ABB RAPID module: TCTM800_DATA.mod

MODULE TCTM800_DATA
    !***********************************************************
    ! Project: P21-100538
    ! Description:
    !   Routines/functions can be modified for the customer
    !
    ! Author: RLZ
    ! Version: 1.0
    ! Date: 04-2022
    !***********************************************************
    !
    !Software axis block
    !Axis 1:                       (-90,-90)
    !Axis 3:                       (-80)
    !
    CONST string sProject:="P21-100538";
    CONST string sScreenMaker:="TpsViewHMI_6700_130220.gtpu.dll";
    !
    CONST num MAX_SPEED:=1000;
    !
    CONST pos WZ_Robot_Home_Box_MIN:=[0,600,1600];
    CONST pos WZ_Robot_Home_Box_MAX:=[800,1600,3000];
    !
    CONST pos WZ_Robot_Inside_Reach_MIN:=[-5000,-5000,-5000];
    CONST pos WZ_Robot_Inside_Reach_MAX:=[15000,5000,5000];
    !
    PERS speeddata vHighSpeed:=[4000,500,150,1000];
    PERS speeddata vHomeBoxSpeed:=[400,80,150,1000];
    PERS speeddata vLowSpeed:=[1000,500,150,1000];
    PERS speeddata vSlowSpeed:=[500,50,150,1000];
    PERS speeddata vSearchSpeed:=[250,500,150,1000];
    PERS speeddata vXsSlowSpeed:=[100,500,150,1000];
    PERS speeddata vXXsSlowSpeed:=[50,500,150,1000];
    !
!    PERS robtarget TargetNew{4000};
    PERS robtarget TargetNew{4000}:=[  [[-19.8208,13.3822,35.1781],[0.985491,-0.093353,0.141246,-0.0119022],[-1,2,-1,1],[6236.68,9E+09,9E+09,9E+09,9E+09,9E+09]],
                                        [[-19.8238,14.3776,34.9882],[0.985491,-0.093353,0.141246,-0.0119022],[-1,2,-1,1],[6236.68,9E+09,9E+09,9E+09,9E+09,9E+09]],
                                        [[-19.8267,15.373,34.7984],[0.985491,-0.093353,0.141246,-0.0119022],[-1,2,-1,1],[6236.68,9E+09,9E+09,9E+09,9E+09,9E+09]],
                                        [[-19.8297,16.3684,34.6085],[0.985491,-0.093353,0.141246,-0.0119022],[-1,2,-1,1],[6236.68,9E+09,9E+09,9E+09,9E+09,9E+09]],
                                        [[-19.8326,17.3638,34.4186],[0.985491,-0.093353,0.141246,-0.0119022],[-1,2,-1,1],[6236.68,9E+09,9E+09,9E+09,9E+09,9E+09]],
                                        [[-19.8356,18.3591,34.2288],[0.985491,-0.093353,0.141246,-0.0119022],[-1,2,-1,1],[6236.68,9E+09,9E+09,9E+09,9E+09,9E+09]],
                                        [[-19.8385,19.3545,34.0389],[0.985491,-0.093353,0.141246,-0.0119022],[-1,2,-1,1],[6236.68,9E+09,9E+09,9E+09,9E+09,9E+09]],
                                        [[-19.8415,20.3499,33.8491],[0.985491,-0.093353,0.141246,-0.0119022],[-1,2,-1,1],[6236.68,9E+09,9E+09,9E+09,9E+09,9E+09]],
                                        [[-19.8444,21.3453,33.6592],[0.985491,-0.093353,0.141246,-0.0119022],[-1,2,-1,1],[6236.68,9E+09,9E+09,9E+09,9E+09,9E+09]],
                                        [[-19.8474,22.3407,33.4694],[0.985491,-0.093353,0.141246,-0.0119022],[-1,2,-1,1],[6236.68,9E+09,9E+09,9E+09,9E+09,9E+09]],
                                        [[-19.8503,23.3361,33.2795],[0.985491,-0.093353,0.141246,-0.0119022],[-1,2,-1,1],[6236.68,9E+09,9E+09,9E+09,9E+09,9E+09]],
                                        [[-19.8533,24.3315,33.0896],[0.985491,-0.093353,0.141246,-0.0119022],[-1,2,-1,1],[6236.68,9E+09,9E+09,9E+09,9E+09,9E+09]],
                                        [[-19.8562,25.3268,32.8998],[0.985491,-0.093353,0.141246,-0.0119022],[-1,2,-1,1],[6236.68,9E+09,9E+09,9E+09,9E+09,9E+09]],
                                        [[-19.8592,26.3222,32.7099],[0.985491,-0.093353,0.141246,-0.0119022],[-1,2,-1,1],[6236.68,9E+09,9E+09,9E+09,9E+09,9E+09]],
                                        [[-19.8621,27.3176,32.5201],[0.985491,-0.093353,0.141246,-0.0119022],[-1,2,-1,1],[6236.68,9E+09,9E+09,9E+09,9E+09,9E+09]],
                                        [[-19.8651,28.313,32.3302],[0.985491,-0.093353,0.141246,-0.0119022],[-1,2,-1,1],[6236.68,9E+09,9E+09,9E+09,9E+09,9E+09]],
                                        [[-19.868,29.3084,32.1403],[0.985491,-0.093353,0.141246,-0.0119022],[-1,2,-1,1],[6236.68,9E+09,9E+09,9E+09,9E+09,9E+09]],
                                        [[-19.871,30.3038,31.9505],[0.985491,-0.093353,0.141246,-0.0119022],[-1,2,-1,1],[6236.68,9E+09,9E+09,9E+09,9E+09,9E+09]],
                                        [[-19.8739,31.2992,31.7606],[0.985491,-0.093353,0.141246,-0.0119022],[-1,2,-1,1],[6236.68,9E+09,9E+09,9E+09,9E+09,9E+09]],
                                        [[-19.8769,32.2945,31.5708],[0.985491,-0.093353,0.141246,-0.0119022],[-1,2,-1,1],[6236.68,9E+09,9E+09,9E+09,9E+09,9E+09]],
                                        [[-19.8798,33.2899,31.3809],[0.985491,-0.093353,0.141246,-0.0119022],[-1,2,-1,1],[6236.68,9E+09,9E+09,9E+09,9E+09,9E+09]],
                                        [[-19.8828,34.2853,31.1911],[0.985491,-0.093353,0.141246,-0.0119022],[-1,2,-1,1],[6236.68,9E+09,9E+09,9E+09,9E+09,9E+09]],
                                        [[-19.8857,35.2807,31.0012],[0.985675,-0.0933685,0.139955,-0.01178],[-1,2,-1,1],[6234.68,9E+09,9E+09,9E+09,9E+09,9E+09]],
                                        [[-19.8887,36.2761,30.8113],[0.985675,-0.0933685,0.139955,-0.01178],[-1,2,-1,1],[6232.68,9E+09,9E+09,9E+09,9E+09,9E+09]],
                                        [[-19.8916,37.2715,30.6215],[0.985675,-0.0933685,0.139955,-0.01178],[-1,2,-1,1],[6230.68,9E+09,9E+09,9E+09,9E+09,9E+09]],
                                        [[-19.8946,38.2669,30.4316],[0.985675,-0.0933685,0.139955,-0.01178],[-1,2,-1,1],[6228.68,9E+09,9E+09,9E+09,9E+09,9E+09]],
                                        [[-19.8976,39.2622,30.2418],[0.985675,-0.0933685,0.139955,-0.01178],[-1,2,-1,1],[6226.68,9E+09,9E+09,9E+09,9E+09,9E+09]],
                                        [[-19.9005,40.2576,30.0519],[0.985675,-0.0933685,0.139955,-0.01178],[-1,2,-1,1],[6224.68,9E+09,9E+09,9E+09,9E+09,9E+09]],
                                        [[-19.9035,41.253,29.8621],[0.985675,-0.0933685,0.139955,-0.01178],[-1,2,-1,1],[6222.68,9E+09,9E+09,9E+09,9E+09,9E+09]],
                                        [[-19.9064,42.2484,29.6722],[0.985675,-0.0933685,0.139955,-0.01178],[-1,2,-1,1],[6220.68,9E+09,9E+09,9E+09,9E+09,9E+09]],
                                        [[-19.9094,43.2438,29.4823],[0.985675,-0.0933685,0.139955,-0.01178],[-1,2,-1,1],[6218.68,9E+09,9E+09,9E+09,9E+09,9E+09]],
                                        [[-19.9123,44.2392,29.2925],[0.985675,-0.0933685,0.139955,-0.01178],[-1,2,-1,1],[6216.68,9E+09,9E+09,9E+09,9E+09,9E+09]],
                                        [[-19.9153,45.2346,29.1026],[0.985675,-0.0933685,0.139955,-0.01178],[-1,2,-1,1],[6214.68,9E+09,9E+09,9E+09,9E+09,9E+09]],
                                        [[-19.9182,46.2299,28.9128],[0.985675,-0.0933685,0.139955,-0.01178],[-1,2,-1,1],[6212.68,9E+09,9E+09,9E+09,9E+09,9E+09]],
                                        [[-19.9212,47.2253,28.7229],[0.985675,-0.0933685,0.139955,-0.01178],[-1,2,-1,1],[6210.68,9E+09,9E+09,9E+09,9E+09,9E+09]],
                                        [[-19.9241,48.2207,28.533],[0.929993,-0.0883232,0.355355,-0.0321736],[-1,2,-1,1],[6212.68,9E+09,9E+09,9E+09,9E+09,9E+09]],
                                        [[-19.9271,49.2161,28.3432],[0.930471,-0.0882227,0.354142,-0.0319903],[-1,2,-1,1],[6214.68,9E+09,9E+09,9E+09,9E+09,9E+09]],
                                        [[-19.93,50.2115,28.1533],[0.930952,-0.0880818,0.352929,-0.031787],[-1,2,-1,1],[6216.68,9E+09,9E+09,9E+09,9E+09,9E+09]],
                                        [[-19.933,51.2069,27.9635],[0.931436,-0.0879018,0.351717,-0.0315633],[-1,2,-1,1],[6218.68,9E+09,9E+09,9E+09,9E+09,9E+09]],
                                        [[-19.9359,52.2022,27.7736],[0.931921,-0.0876857,0.350504,-0.0313225],[-1,2,-1,1],[6220.68,9E+09,9E+09,9E+09,9E+09,9E+09]],
                                        [[-19.9389,53.1976,27.5838],[0.932407,-0.0874409,0.349293,-0.0310697],[-1,2,-1,1],[6222.68,9E+09,9E+09,9E+09,9E+09,9E+09]],
                                        [[-19.9418,54.193,27.3939],[0.932894,-0.0871662,0.348081,-0.0308115],[-1,2,-1,1],[6224.68,9E+09,9E+09,9E+09,9E+09,9E+09]],
                                        [[-19.9448,55.1884,27.204],[0.933381,-0.0868686,0.346871,-0.0305526],[-1,2,-1,1],[6226.68,9E+09,9E+09,9E+09,9E+09,9E+09]],
                                        [[-19.9477,56.1838,27.0142],[0.933868,-0.0865579,0.34566,-0.0302899],[-1,2,-1,1],[6228.68,9E+09,9E+09,9E+09,9E+09,9E+09]],
                                        [[-19.9507,57.1792,26.8243],[0.934353,-0.0862461,0.344448,-0.0300257],[-1,2,-1,1],[6230.68,9E+09,9E+09,9E+09,9E+09,9E+09]],
                                        [[-19.9536,58.1746,26.6345],[0.934837,-0.0859295,0.343235,-0.0297506],[-1,2,-1,1],[6232.68,9E+09,9E+09,9E+09,9E+09,9E+09]],
                                        [[-19.9566,59.1699,26.4446],[0.93532,-0.0856102,0.342021,-0.0294673],[-1,2,-1,1],[6234.68,9E+09,9E+09,9E+09,9E+09,9E+09]],
                                        [[-19.9595,60.1653,26.2548],[0.935802,-0.0852947,0.340805,-0.0291789],[-1,2,-1,1],[6236.68,9E+09,9E+09,9E+09,9E+09,9E+09]],
                                        [[-19.9625,61.1607,26.0649],[0.936281,-0.0849877,0.339588,-0.0288886],[-1,2,-1,1],[6238.68,9E+09,9E+09,9E+09,9E+09,9E+09]],
                                        [[-19.9654,62.1561,25.875],[0.936758,-0.0846954,0.33837,-0.0285976],[-1,2,-1,1],[6240.68,9E+09,9E+09,9E+09,9E+09,9E+09]],
                                        [[-19.9684,63.1515,25.6852],[0.937231,-0.0844174,0.33715,-0.0283113],[-1,2,-1,1],[6242.68,9E+09,9E+09,9E+09,9E+09,9E+09]],
                                        [[-19.9713,64.1469,25.4953],[0.937701,-0.0841591,0.335928,-0.0280356],[-1,2,-1,1],[6244.68,9E+09,9E+09,9E+09,9E+09,9E+09]],
                                        [[-19.9792,65.5555,25.2738],[0.938167,-0.0839191,0.334706,-0.0277747],[-1,2,-1,1],[6246.68,9E+09,9E+09,9E+09,9E+09,9E+09]],
                                        [[-19.9846,66.7312,25.0742],[0.938629,-0.0837057,0.333483,-0.0275222],[-1,2,-1,1],[6248.68,9E+09,9E+09,9E+09,9E+09,9E+09]],
                                        [[-19.9903,67.8868,24.8779],[0.939087,-0.0835199,0.332257,-0.0272796],[-1,2,-1,1],[6250.68,9E+09,9E+09,9E+09,9E+09,9E+09]],
                                        [[-19.9968,69.025,24.6862],[0.939537,-0.0834029,0.33103,-0.0270736],[-1,2,-1,1],[6252.68,9E+09,9E+09,9E+09,9E+09,9E+09]],
                                        [[-20.0023,70.1507,24.4974],[0.939978,-0.0833611,0.3298,-0.0269014],[-1,2,-1,1],[6254.68,9E+09,9E+09,9E+09,9E+09,9E+09]],
                                        [[-20.0074,71.2662,24.3079],[0.940411,-0.0833921,0.328567,-0.026763],[-1,2,-1,1],[6256.68,9E+09,9E+09,9E+09,9E+09,9E+09]],
                                        [[-20.0097,72.3751,24.121],[0.940835,-0.0835,0.327332,-0.0266604],[-1,2,-1,1],[6258.68,9E+09,9E+09,9E+09,9E+09,9E+09]],
                                        [[-20.0112,73.4816,23.9325],[0.94125,-0.0836821,0.326095,-0.0265903],[-1,2,-1,1],[6260.68,9E+09,9E+09,9E+09,9E+09,9E+09]],
                                        [[-20.0151,74.5864,23.7424],[0.941657,-0.0839444,0.324855,-0.0265527],[-1,2,-1,1],[6262.68,9E+09,9E+09,9E+09,9E+09,9E+09]],
                                        [[-20.0203,75.6949,23.5472],[0.942055,-0.0842785,0.323612,-0.0265474],[-1,2,-1,1],[6264.68,9E+09,9E+09,9E+09,9E+09,9E+09]],
                                        [[-20.0287,76.8065,23.3556],[0.942445,-0.084682,0.322367,-0.0265724],[-1,2,-1,1],[6266.68,9E+09,9E+09,9E+09,9E+09,9E+09]],
                                        [[-20.0368,77.9219,23.1634],[0.942828,-0.0851371,0.321121,-0.0266187],[-1,2,-1,1],[6268.68,9E+09,9E+09,9E+09,9E+09,9E+09]],
                                        [[-20.0447,79.0403,22.9681],[0.943204,-0.0856504,0.319872,-0.0266856],[-1,2,-1,1],[6270.68,9E+09,9E+09,9E+09,9E+09,9E+09]],
                                        [[-20.0527,80.1618,22.7711],[0.943573,-0.0862256,0.31862,-0.0267765],[-1,2,-1,1],[6272.68,9E+09,9E+09,9E+09,9E+09,9E+09]],
                                        [[-20.0612,81.2846,22.5719],[0.943932,-0.0868722,0.317367,-0.0269036],[-1,2,-1,1],[6274.68,9E+09,9E+09,9E+09,9E+09,9E+09]],
                                        [[-20.0679,82.4167,22.3707],[0.944282,-0.0875917,0.316112,-0.0270609],[-1,2,-1,1],[6276.68,9E+09,9E+09,9E+09,9E+09,9E+09]],
                                        [[-20.0726,83.5525,22.1667],[0.944623,-0.0883798,0.314854,-0.0272472],[-1,2,-1,1],[6278.68,9E+09,9E+09,9E+09,9E+09,9E+09]],
                                        [[-20.0759,84.6909,21.9623],[0.944955,-0.0892357,0.313595,-0.027466],[-1,2,-1,1],[6280.49,9E+09,9E+09,9E+09,9E+09,9E+09]],
                                        [[-20.0829,85.8322,21.7552],[0.945292,-0.090032,0.312336,-0.0276392],[-1,2,-1,1],[6282.04,9E+09,9E+09,9E+09,9E+09,9E+09]],
                                        [[-20.0895,86.9766,21.5476],[0.94563,-0.0908122,0.311073,-0.0277661],[-1,2,-1,1],[6283.36,9E+09,9E+09,9E+09,9E+09,9E+09]],
                                        [[-20.09,87.9047,21.3558],[0.94597,-0.0915639,0.309808,-0.0278434],[-1,2,-1,1],[6284.46,9E+09,9E+09,9E+09,9E+09,9E+09]],
                                        [[-20.0924,88.8463,21.1574],[0.946315,-0.0922771,0.30854,-0.0278587],[-1,2,-1,1],[6285.55,9E+09,9E+09,9E+09,9E+09,9E+09]],
                                        [[-20.0944,89.8013,20.9561],[0.946663,-0.0929378,0.307272,-0.0278381],[-1,2,-1,1],[6286.4,9E+09,9E+09,9E+09,9E+09,9E+09]],
                                        [[-20.0959,90.781,20.7473],[0.947015,-0.0935522,0.306003,-0.0277818],[-1,2,-1,1],[6287.04,9E+09,9E+09,9E+09,9E+09,9E+09]],
                                        [[-20.0983,91.779,20.5356],[0.947371,-0.0941184,0.304734,-0.027689],[-1,2,-1,1],[6287.46,9E+09,9E+09,9E+09,9E+09,9E+09]],
                                        [[-20.1012,92.7833,20.3188],[0.947729,-0.0946464,0.303465,-0.0275732],[-1,2,-1,1],[6287.67,9E+09,9E+09,9E+09,9E+09,9E+09]],
                                        [[-20.1031,93.793,20.1035],[0.94809,-0.0951344,0.302195,-0.0274276],[-1,2,-1,1],[6287.7,9E+09,9E+09,9E+09,9E+09,9E+09]],
                                        [[-20.1053,94.8139,19.887],[0.948456,-0.0955701,0.300925,-0.0272494],[-1,2,-1,1],[6287.54,9E+09,9E+09,9E+09,9E+09,9E+09]],
                                        [[-20.1085,95.8306,19.6795],[0.948826,-0.0959528,0.299654,-0.0270214],[-1,2,-1,1],[6287.21,9E+09,9E+09,9E+09,9E+09,9E+09]],
                                        [[-20.113,96.8463,19.469],[0.949202,-0.0962697,0.298382,-0.026743],[-1,2,-1,1],[6286.72,9E+09,9E+09,9E+09,9E+09,9E+09]],
                                        [[-20.1163,97.8528,19.258],[0.949586,-0.0965149,0.297109,-0.0264101],[-1,2,-1,1],[6286.07,9E+09,9E+09,9E+09,9E+09,9E+09]],
                                        [[-20.1158,98.8519,19.0415],[0.949976,-0.0966895,0.295836,-0.0260264],[-1,2,-1,1],[6285.28,9E+09,9E+09,9E+09,9E+09,9E+09]],
                                        [[-20.118,99.846,18.8262],[0.950371,-0.0968106,0.294562,-0.0255972],[-1,2,-1,1],[6284.35,9E+09,9E+09,9E+09,9E+09,9E+09]],
                                        [[-20.1194,100.834,18.6136],[0.950772,-0.0968625,0.293289,-0.0251351],[-1,2,-1,1],[6283.29,9E+09,9E+09,9E+09,9E+09,9E+09]],
                                        [[-20.1198,101.816,18.4019],[0.95118,-0.0968264,0.292018,-0.0246466],[-1,2,-1,1],[6282.1,9E+09,9E+09,9E+09,9E+09,9E+09]],
                                        [[-20.132,102.941,18.1808],[0.951594,-0.0967003,0.290751,-0.0241347],[-1,2,-1,1],[6280.79,9E+09,9E+09,9E+09,9E+09,9E+09]],
                                        [[-20.1525,104.034,17.9652],[0.952015,-0.0964822,0.289486,-0.0236033],[-1,2,-1,1],[6279.23,9E+09,9E+09,9E+09,9E+09,9E+09]],
                                        [[-20.1727,105.104,17.7578],[0.952442,-0.096171,0.288226,-0.0230543],[-1,2,-1,1],[6277.6,9E+09,9E+09,9E+09,9E+09,9E+09]],
                                        [[-20.1965,106.149,17.558],[0.95287,-0.0958206,0.286967,-0.0225081],[-1,2,-1,1],[6275.89,9E+09,9E+09,9E+09,9E+09,9E+09]],
                                        [[-20.2098,107.165,17.3633],[0.953295,-0.0954673,0.285711,-0.0219992],[-1,2,-1,1],[6274.12,9E+09,9E+09,9E+09,9E+09,9E+09]],
                                        [[-20.2242,108.185,17.1667],[0.953715,-0.0951127,0.284459,-0.0215388],[-1,2,-1,1],[6272.29,9E+09,9E+09,9E+09,9E+09,9E+09]],
                                        [[-20.2425,109.218,16.9643],[0.954131,-0.0947572,0.28321,-0.0211306],[-1,2,-1,1],[6270.39,9E+09,9E+09,9E+09,9E+09,9E+09]],
                                        [[-20.2581,110.254,16.7562],[0.954543,-0.0944062,0.281965,-0.0207777],[-1,2,-1,1],[6268.41,9E+09,9E+09,9E+09,9E+09,9E+09]],
                                        [[-20.2753,111.299,16.547],[0.954949,-0.0940667,0.280722,-0.0204648],[-1,2,-1,1],[6266.41,9E+09,9E+09,9E+09,9E+09,9E+09]],
                                        [[-20.2912,112.342,16.3468],[0.955352,-0.09373,0.279481,-0.0201944],[-1,2,-1,1],[6264.41,9E+09,9E+09,9E+09,9E+09,9E+09]],
                                        [[-20.3116,113.385,16.1428],[0.955753,-0.0933758,0.278243,-0.0199595],[-1,2,-1,1],[6262.41,9E+09,9E+09,9E+09,9E+09,9E+09]],
                                        [[-20.3318,114.437,15.9409],[0.956155,-0.0929712,0.27701,-0.0197528],[-1,2,-1,1],[6260.41,9E+09,9E+09,9E+09,9E+09,9E+09]],
                                        [[-20.3539,115.497,15.7419],[0.956556,-0.0925336,0.275781,-0.0195746],[-1,2,-1,1],[6258.41,9E+09,9E+09,9E+09,9E+09,9E+09]],
                                        [[-20.376,116.553,15.5421],[0.956956,-0.0920778,0.274554,-0.0194295],[-1,2,-1,1],[6256.41,9E+09,9E+09,9E+09,9E+09,9E+09]],
                                        [[-20.3986,117.615,15.334],[0.957352,-0.0916118,0.273332,-0.0193503],[-1,2,-1,1],[6254.41,9E+09,9E+09,9E+09,9E+09,9E+09]],
                                        [[-20.4172,118.682,15.1287],[0.957744,-0.0911493,0.272113,-0.0193238],[-1,2,-1,1],[6252.41,9E+09,9E+09,9E+09,9E+09,9E+09]],
                                        [[-20.4343,119.758,14.9301],[0.958131,-0.0906871,0.270898,-0.0193504],[-1,2,-1,1],[6250.41,9E+09,9E+09,9E+09,9E+09,9E+09]],
                                        [[-20.4523,120.845,14.7299],[0.958515,-0.0902277,0.269686,-0.0194368],[-1,2,-1,1],[6248.41,9E+09,9E+09,9E+09,9E+09,9E+09]],
                                        [[-20.4663,121.94,14.5304],[0.958898,-0.089739,0.268477,-0.0195467],[-1,2,-1,1],[6246.41,9E+09,9E+09,9E+09,9E+09,9E+09]],
                                        [[-20.4807,123.047,14.3291],[0.959282,-0.0892157,0.267268,-0.0196568],[-1,2,-1,1],[6244.41,9E+09,9E+09,9E+09,9E+09,9E+09]],
                                        [[-20.4981,124.154,14.1317],[0.959667,-0.0886629,0.266059,-0.0197558],[-1,2,-1,1],[6242.41,9E+09,9E+09,9E+09,9E+09,9E+09]],
                                        [[-20.5026,125.121,13.9475],[0.960055,-0.0880643,0.26485,-0.0198288],[-1,2,-1,1],[6240.41,9E+09,9E+09,9E+09,9E+09,9E+09]],
                                        [[-20.5034,126.11,13.7579],[0.960445,-0.087429,0.263639,-0.0198882],[-1,2,-1,1],[6238.41,9E+09,9E+09,9E+09,9E+09,9E+09]],
                                        [[-20.5034,127.127,13.5658],[0.960836,-0.0867591,0.262429,-0.0199342],[-1,2,-1,1],[6236.41,9E+09,9E+09,9E+09,9E+09,9E+09]],
                                        [[-20.5024,128.169,13.3659],[0.961228,-0.0860689,0.261217,-0.0199642],[-1,2,-1,1],[6234.41,9E+09,9E+09,9E+09,9E+09,9E+09]],
                                        [[-20.5079,129.246,13.1642],[0.961619,-0.0853668,0.260003,-0.0199849],[-1,2,-1,1],[6232.41,9E+09,9E+09,9E+09,9E+09,9E+09]],
                                        [[-20.5129,130.318,12.9654],[0.96201,-0.0846451,0.258789,-0.0200034],[-1,2,-1,1],[6230.41,9E+09,9E+09,9E+09,9E+09,9E+09]],
                                        [[-20.5176,131.386,12.7781],[0.962402,-0.0838952,0.257574,-0.0200107],[-1,2,-1,1],[6228.41,9E+09,9E+09,9E+09,9E+09,9E+09]],
                                        [[-20.521,132.452,12.6002],[0.962793,-0.083134,0.256357,-0.0199986],[-1,2,-1,1],[6226.41,9E+09,9E+09,9E+09,9E+09,9E+09]],
                                        [[-20.5242,133.524,12.4195],[0.963184,-0.0823558,0.255137,-0.0199609],[-1,2,-1,1],[6224.41,9E+09,9E+09,9E+09,9E+09,9E+09]],
                                        [[-20.529,134.597,12.236],[0.963577,-0.0815547,0.253915,-0.0198901],[-1,2,-1,1],[6222.41,9E+09,9E+09,9E+09,9E+09,9E+09]],
                                        [[-20.5243,135.676,12.0539],[0.963969,-0.0807422,0.25269,-0.019793],[-1,2,-1,1],[6220.41,9E+09,9E+09,9E+09,9E+09,9E+09]],
                                        [[-20.5241,136.752,11.8701],[0.964361,-0.0799295,0.251461,-0.0196632],[-1,2,-1,1],[6218.41,9E+09,9E+09,9E+09,9E+09,9E+09]],
                                        [[-20.5233,137.834,11.6876],[0.964753,-0.0791039,0.250229,-0.0195004],[-1,2,-1,1],[6216.41,9E+09,9E+09,9E+09,9E+09,9E+09]],
                                        [[-20.5213,138.917,11.5061],[0.965145,-0.0782514,0.248995,-0.0193104],[-1,2,-1,1],[6214.41,9E+09,9E+09,9E+09,9E+09,9E+09]],
                                        [[-20.5195,140.009,11.3264],[0.965539,-0.0773669,0.247759,-0.0190841],[-1,2,-1,1],[6212.41,9E+09,9E+09,9E+09,9E+09,9E+09]],
                                        [[-20.5177,141.101,11.1547],[0.965934,-0.0764373,0.246522,-0.0188431],[-1,2,-1,1],[6210.41,9E+09,9E+09,9E+09,9E+09,9E+09]],
                                        [[-20.5194,142.191,10.9814],[0.96633,-0.0754803,0.245284,-0.0185802],[-1,2,-1,1],[6208.41,9E+09,9E+09,9E+09,9E+09,9E+09]],
                                        [[-20.5206,143.275,10.8171],[0.966726,-0.0744976,0.244042,-0.018276],[-1,2,-1,1],[6206.41,9E+09,9E+09,9E+09,9E+09,9E+09]],
                                        [[-20.5271,144.346,10.6525],[0.96712,-0.0735062,0.2428,-0.0179729],[-1,2,-1,1],[6204.41,9E+09,9E+09,9E+09,9E+09,9E+09]],
                                        [[-20.5322,145.413,10.491],[0.967512,-0.0725173,0.241557,-0.0176804],[-1,2,-1,1],[6202.41,9E+09,9E+09,9E+09,9E+09,9E+09]],
                                        [[-20.5358,146.488,10.3282],[0.9679,-0.0715185,0.240314,-0.017403],[-1,2,-1,1],[6200.41,9E+09,9E+09,9E+09,9E+09,9E+09]],
                                        [[-20.5395,147.562,10.1691],[0.968285,-0.0705347,0.239071,-0.0171473],[-1,2,-1,1],[6198.41,9E+09,9E+09,9E+09,9E+09,9E+09]],
                                        [[-20.5371,148.636,10.0155],[0.968666,-0.0695557,0.237828,-0.0169132],[-1,2,-1,1],[6196.41,9E+09,9E+09,9E+09,9E+09,9E+09]],
                                        [[-20.5375,149.7,9.86272],[0.969044,-0.0685852,0.236584,-0.0166887],[-1,2,-1,1],[6194.41,9E+09,9E+09,9E+09,9E+09,9E+09]],
                                        [[-20.5382,150.759,9.71114],[0.969419,-0.0676025,0.23534,-0.0164729],[-1,2,-1,1],[6192.41,9E+09,9E+09,9E+09,9E+09,9E+09]],
                                        [[-20.5401,151.807,9.56385],[0.969793,-0.0666008,0.234096,-0.0162691],[-1,2,-1,1],[6190.41,9E+09,9E+09,9E+09,9E+09,9E+09]],
                                        [[-20.5411,152.853,9.41893],[0.970165,-0.0655904,0.232851,-0.0160605],[-1,2,-1,1],[6188.41,9E+09,9E+09,9E+09,9E+09,9E+09]],
                                        [[-20.5401,153.892,9.27389],[0.970534,-0.0645924,0.231603,-0.0158409],[-1,2,-1,1],[6186.41,9E+09,9E+09,9E+09,9E+09,9E+09]],
                                        [[-20.5407,154.936,9.13387],[0.9709,-0.0635957,0.230355,-0.0156395],[-1,2,-1,1],[6184.41,9E+09,9E+09,9E+09,9E+09,9E+09]],
                                        [[-20.5431,155.978,8.99994],[0.971262,-0.0626252,0.229107,-0.015458],[-1,2,-1,1],[6182.41,9E+09,9E+09,9E+09,9E+09,9E+09]],
                                        [[-20.5425,157.019,8.86639],[0.971619,-0.0616734,0.227858,-0.0152985],[-1,2,-1,1],[6180.41,9E+09,9E+09,9E+09,9E+09,9E+09]],
                                        [[-20.5431,158.057,8.74051],[0.971972,-0.0607409,0.226608,-0.0151596],[-1,2,-1,1],[6178.41,9E+09,9E+09,9E+09,9E+09,9E+09]],
                                        [[-20.5359,159.087,8.62099],[0.972321,-0.0598333,0.225358,-0.0150446],[-1,2,-1,1],[6176.41,9E+09,9E+09,9E+09,9E+09,9E+09]],
                                        [[-20.5325,160.108,8.49936],[0.972666,-0.058934,0.224107,-0.0149464],[-1,2,-1,1],[6174.41,9E+09,9E+09,9E+09,9E+09,9E+09]],
                                        [[-20.5335,161.122,8.38014],[0.973008,-0.058059,0.222856,-0.0148563],[-1,2,-1,1],[6172.43,9E+09,9E+09,9E+09,9E+09,9E+09]],
                                        [[-20.5305,162.119,8.26332],[0.973347,-0.0571837,0.221603,-0.0147792],[-1,2,-1,1],[6170.5,9E+09,9E+09,9E+09,9E+09,9E+09]],
                                        [[-20.5281,163.112,8.14692],[0.973683,-0.0563282,0.220349,-0.0146903],[-1,2,-1,1],[6168.61,9E+09,9E+09,9E+09,9E+09,9E+09]],
                                        [[-20.5233,164.107,8.03679],[0.974016,-0.0554899,0.219093,-0.014597],[-1,2,-1,1],[6166.75,9E+09,9E+09,9E+09,9E+09,9E+09]],
                                        [[-20.5187,165.099,7.92401],[0.974345,-0.054675,0.217835,-0.0145069],[-1,2,-1,1],[6164.91,9E+09,9E+09,9E+09,9E+09,9E+09]],
                                        [[-20.5066,166.097,7.81529],[0.974672,-0.0538733,0.216576,-0.0144121],[-1,2,-1,1],[6163.09,9E+09,9E+09,9E+09,9E+09,9E+09]],
                                        [[-20.4993,167.094,7.70887],[0.974996,-0.053085,0.215315,-0.0143165],[-1,2,-1,1],[6161.29,9E+09,9E+09,9E+09,9E+09,9E+09]],
                                        [[-20.4897,168.086,7.60563],[0.975316,-0.0523195,0.214053,-0.014217],[-1,2,-1,1],[6159.52,9E+09,9E+09,9E+09,9E+09,9E+09]],
                                        [[-20.4792,169.072,7.49978],[0.975634,-0.0515742,0.212789,-0.0141096],[-1,2,-1,1],[6157.76,9E+09,9E+09,9E+09,9E+09,9E+09]],
                                        [[-20.476,170.058,7.39684],[0.975949,-0.0508484,0.211524,-0.0139848],[-1,2,-1,1],[6156.03,9E+09,9E+09,9E+09,9E+09,9E+09]],
                                        [[-20.4754,171.047,7.29169],[0.976262,-0.05014,0.210256,-0.0138475],[-1,2,-1,1],[6154.31,9E+09,9E+09,9E+09,9E+09,9E+09]],
                                        [[-20.4712,172.039,7.18915],[0.976571,-0.0494588,0.208987,-0.013702],[-1,2,-1,1],[6152.6,9E+09,9E+09,9E+09,9E+09,9E+09]],
                                        [[-20.4641,173.037,7.08129],[0.976877,-0.0487983,0.207716,-0.0135442],[-1,2,-1,1],[6150.89,9E+09,9E+09,9E+09,9E+09,9E+09]],
                                        [[-20.4553,174.038,6.97779],[0.977182,-0.0481431,0.206444,-0.0133751],[-1,2,-1,1],[6149.18,9E+09,9E+09,9E+09,9E+09,9E+09]],
                                        [[-20.4481,175.039,6.8771],[0.977484,-0.0474869,0.205171,-0.0132028],[-1,2,-1,1],[6147.48,9E+09,9E+09,9E+09,9E+09,9E+09]],
                                        [[-20.4396,176.048,6.7746],[0.977785,-0.046821,0.203897,-0.0130177],[-1,2,-1,1],[6145.79,9E+09,9E+09,9E+09,9E+09,9E+09]],
                                        [[-20.4321,177.052,6.67588],[0.978086,-0.0461204,0.202622,-0.0128224],[-1,2,-1,1],[6144.09,9E+09,9E+09,9E+09,9E+09,9E+09]],
                                        [[-20.4253,178.052,6.57796],[0.978386,-0.0454033,0.201346,-0.01261],[-1,2,-1,1],[6142.42,9E+09,9E+09,9E+09,9E+09,9E+09]],
                                        [[-20.4145,179.05,6.48497],[0.978685,-0.0446681,0.200069,-0.0123735],[-1,2,-1,1],[6140.75,9E+09,9E+09,9E+09,9E+09,9E+09]],
                                        [[-20.4095,180.058,6.39117],[0.978982,-0.0439253,0.198791,-0.0121204],[-1,2,-1,1],[6139.1,9E+09,9E+09,9E+09,9E+09,9E+09]],
                                        [[-20.4019,181.065,6.29868],[0.979278,-0.043166,0.197512,-0.0118629],[-1,2,-1,1],[6137.44,9E+09,9E+09,9E+09,9E+09,9E+09]],
                                        [[-20.3919,182.079,6.20642],[0.979572,-0.0423833,0.196233,-0.0115968],[-1,2,-1,1],[6135.79,9E+09,9E+09,9E+09,9E+09,9E+09]],
                                        [[-20.3839,183.106,6.11795],[0.979865,-0.0416076,0.194952,-0.0113066],[-1,2,-1,1],[6134.15,9E+09,9E+09,9E+09,9E+09,9E+09]],
                                        [[-20.3794,184.135,6.02731],[0.980155,-0.040822,0.19367,-0.0110132],[-1,2,-1,1],[6132.5,9E+09,9E+09,9E+09,9E+09,9E+09]],
                                        [[-20.3739,185.17,5.93653],[0.980444,-0.0400121,0.192388,-0.0107093],[-1,2,-1,1],[6130.85,9E+09,9E+09,9E+09,9E+09,9E+09]],
                                        [[-20.3693,186.202,5.85017],[0.980732,-0.0391786,0.191105,-0.0103939],[-1,2,-1,1],[6129.21,9E+09,9E+09,9E+09,9E+09,9E+09]],
                                        [[-20.367,187.237,5.76598],[0.981018,-0.0383365,0.189821,-0.0100737],[-1,2,-1,1],[6127.58,9E+09,9E+09,9E+09,9E+09,9E+09]],
                                        [[-20.3627,188.275,5.68342],[0.981302,-0.0374851,0.188537,-0.00974249],[-1,2,-1,1],[6125.96,9E+09,9E+09,9E+09,9E+09,9E+09]],
                                        [[-20.3598,189.315,5.60034],[0.981584,-0.0366277,0.187252,-0.0093854],[-1,2,-1,1],[6124.35,9E+09,9E+09,9E+09,9E+09,9E+09]],
                                        [[-20.3555,190.358,5.51843],[0.981864,-0.0357578,0.185966,-0.00902299],[-1,2,-1,1],[6122.74,9E+09,9E+09,9E+09,9E+09,9E+09]],
                                        [[-20.3476,191.416,5.43901],[0.982141,-0.0348906,0.184679,-0.0086603],[-1,2,-1,1],[6121.14,9E+09,9E+09,9E+09,9E+09,9E+09]],
                                        [[-20.3383,192.469,5.36491],[0.982416,-0.034018,0.183393,-0.00830042],[-1,2,-1,1],[6119.53,9E+09,9E+09,9E+09,9E+09,9E+09]],
                                        [[-20.3303,193.528,5.29109],[0.982688,-0.0331399,0.182106,-0.00793952],[-1,2,-1,1],[6117.94,9E+09,9E+09,9E+09,9E+09,9E+09]],
                                        [[-20.3271,194.59,5.22459],[0.982958,-0.0322531,0.180819,-0.00758491],[-1,2,-1,1],[6116.36,9E+09,9E+09,9E+09,9E+09,9E+09]],
                                        [[-20.3244,195.653,5.15782],[0.983226,-0.0313631,0.179531,-0.00723374],[-1,2,-1,1],[6114.79,9E+09,9E+09,9E+09,9E+09,9E+09]],
                                        [[-20.3202,196.718,5.09376],[0.98349,-0.0304714,0.178244,-0.00688634],[-1,2,-1,1],[6113.23,9E+09,9E+09,9E+09,9E+09,9E+09]],
                                        [[-20.3179,197.777,5.02838],[0.983753,-0.0295701,0.176956,-0.00654743],[-1,2,-1,1],[6111.68,9E+09,9E+09,9E+09,9E+09,9E+09]],
                                        [[-20.3094,198.839,4.9687],[0.984012,-0.0286624,0.175668,-0.00621116],[-1,2,-1,1],[6110.16,9E+09,9E+09,9E+09,9E+09,9E+09]],
                                        [[-20.3041,199.901,4.90933],[0.98427,-0.0277469,0.174381,-0.00588522],[-1,2,-1,1],[6108.65,9E+09,9E+09,9E+09,9E+09,9E+09]],
                                        [[-20.3079,200.963,4.845],[0.984524,-0.0268254,0.173093,-0.00557557],[-1,2,-1,1],[6107.16,9E+09,9E+09,9E+09,9E+09,9E+09]],
                                        [[-20.3097,202.026,4.78401],[0.984777,-0.0258792,0.171805,-0.00527546],[-1,2,-1,1],[6105.69,9E+09,9E+09,9E+09,9E+09,9E+09]],
                                        [[-20.3096,203.096,4.73043],[0.985026,-0.02494,0.170517,-0.00497303],[-1,2,-1,1],[6104.24,9E+09,9E+09,9E+09,9E+09,9E+09]],
                                        [[-20.3123,204.167,4.67704],[0.985273,-0.0240038,0.169229,-0.00467442],[-1,2,-1,1],[6102.8,9E+09,9E+09,9E+09,9E+09,9E+09]],
                                        [[-20.316,205.234,4.62361],[0.985518,-0.0230589,0.16794,-0.00438433],[-1,2,-1,1],[6101.39,9E+09,9E+09,9E+09,9E+09,9E+09]],
                                        [[-20.3149,206.309,4.57073],[0.98576,-0.0221061,0.166651,-0.00409394],[-1,2,-1,1],[6100,9E+09,9E+09,9E+09,9E+09,9E+09]],
                                        [[-20.3178,207.379,4.52344],[0.985999,-0.0211567,0.165362,-0.00380563],[-1,2,-1,1],[6098.62,9E+09,9E+09,9E+09,9E+09,9E+09]],
                                        [[-20.3159,208.454,4.47764],[0.986235,-0.0202181,0.164072,-0.003527],[-1,2,-1,1],[6097.28,9E+09,9E+09,9E+09,9E+09,9E+09]],
                                        [[-20.316,209.53,4.4335],[0.986468,-0.0192851,0.162782,-0.00326316],[-1,2,-1,1],[6095.95,9E+09,9E+09,9E+09,9E+09,9E+09]],
                                        [[-20.3165,210.598,4.39223],[0.986699,-0.0183481,0.161493,-0.0030208],[-1,2,-1,1],[6094.64,9E+09,9E+09,9E+09,9E+09,9E+09]],
                                        [[-20.3171,211.668,4.35232],[0.986927,-0.0174043,0.160203,-0.00281226],[-1,2,-1,1],[6093.38,9E+09,9E+09,9E+09,9E+09,9E+09]],
                                        [[-20.3166,212.738,4.31818],[0.987152,-0.0164551,0.158914,-0.0026257],[-1,2,-1,1],[6092.13,9E+09,9E+09,9E+09,9E+09,9E+09]],
                                        [[-20.3168,213.797,4.28298],[0.987375,-0.0154957,0.157624,-0.00245473],[-1,2,-1,1],[6090.92,9E+09,9E+09,9E+09,9E+09,9E+09]],
                                        [[-20.3168,214.866,4.24987],[0.987595,-0.0145298,0.156334,-0.00230076],[-1,2,-1,1],[6089.76,9E+09,9E+09,9E+09,9E+09,9E+09]],
                                        [[-20.319,215.931,4.21878],[0.987812,-0.013548,0.155044,-0.00216247],[-1,2,-1,1],[6088.61,9E+09,9E+09,9E+09,9E+09,9E+09]],
                                        [[-20.3184,216.989,4.19102],[0.988027,-0.0125584,0.153753,-0.00203146],[-1,2,-1,1],[6087.51,9E+09,9E+09,9E+09,9E+09,9E+09]],
                                        [[-20.3174,218.042,4.16606],[0.98824,-0.0115488,0.152462,-0.00192143],[-1,2,-1,1],[6086.45,9E+09,9E+09,9E+09,9E+09,9E+09]],
                                        [[-20.3166,219.099,4.14279],[0.98845,-0.0105256,0.151171,-0.00183378],[-1,2,-1,1],[6085.44,9E+09,9E+09,9E+09,9E+09,9E+09]],
                                        [[-20.3159,220.152,4.12782],[0.988657,-0.00950032,0.149879,-0.00175203],[-1,2,-1,1],[6084.46,9E+09,9E+09,9E+09,9E+09,9E+09]],
                                        [[-20.3194,221.196,4.10654],[0.988862,-0.00847964,0.148587,-0.00168042],[-1,2,-1,1],[6083.52,9E+09,9E+09,9E+09,9E+09,9E+09]],
                                        [[-20.3215,222.236,4.0906],[0.989063,-0.00744996,0.147294,-0.00161937],[-1,2,-1,1],[6082.63,9E+09,9E+09,9E+09,9E+09,9E+09]],
                                        [[-20.3201,223.276,4.07881],[0.989263,-0.00641868,0.146,-0.00156027],[-1,2,-1,1],[6081.78,9E+09,9E+09,9E+09,9E+09,9E+09]],
                                        [[-20.3203,224.318,4.06922],[0.989459,-0.00539295,0.144706,-0.00149868],[-1,2,-1,1],[6080.97,9E+09,9E+09,9E+09,9E+09,9E+09]],
                                        [[-20.3226,225.354,4.05679],[0.989653,-0.00437349,0.143411,-0.00145052],[-1,2,-1,1],[6080.19,9E+09,9E+09,9E+09,9E+09,9E+09]],
                                        [[-20.3212,226.401,4.04463],[0.989843,-0.00335394,0.142116,-0.00140343],[-1,2,-1,1],[6079.45,9E+09,9E+09,9E+09,9E+09,9E+09]],
                                        [[-20.3183,227.448,4.03686],[0.990032,-0.0023352,0.14082,-0.00136396],[-1,2,-1,1],[6078.74,9E+09,9E+09,9E+09,9E+09,9E+09]],
                                        [[-20.3156,228.491,4.03409],[0.990217,-0.00132889,0.139523,-0.00133138],[-1,2,-1,1],[6078.06,9E+09,9E+09,9E+09,9E+09,9E+09]],
                                        [[-20.3097,229.531,4.03064],[0.9904,-0.000318447,0.138226,-0.00130941],[-1,2,-1,1],[6077.43,9E+09,9E+09,9E+09,9E+09,9E+09]],
                                        [[-20.3073,230.568,4.03131],[0.99058,0.000703247,0.136928,-0.00129069],[-1,2,-1,1],[6079.43,9E+09,9E+09,9E+09,9E+09,9E+09]],
                                        [[-20.303,231.603,4.0306],[0.990757,0.00174002,0.135629,-0.00127438],[-1,2,-1,1],[6081.43,9E+09,9E+09,9E+09,9E+09,9E+09]],
                                        [[-20.2976,232.639,4.0324],[0.990932,0.00278063,0.13433,-0.00126001],[-1,2,-1,1],[6083.43,9E+09,9E+09,9E+09,9E+09,9E+09]],
                                        [[-20.2937,233.675,4.03945],[0.991104,0.00382398,0.13303,-0.00124399],[-1,2,-1,1],[6085.43,9E+09,9E+09,9E+09,9E+09,9E+09]],
                                        [[-20.2921,234.71,4.04898],[0.991273,0.00486029,0.13173,-0.00121866],[-1,2,-1,1],[6087.43,9E+09,9E+09,9E+09,9E+09,9E+09]],
                                        [[-20.2901,235.745,4.06115],[0.991439,0.00589237,0.130429,-0.00119014],[-1,2,-1,1],[6089.43,9E+09,9E+09,9E+09,9E+09,9E+09]],
                                        [[-20.2852,236.773,4.07455],[0.991603,0.00692863,0.129128,-0.00116419],[-1,2,-1,1],[6091.43,9E+09,9E+09,9E+09,9E+09,9E+09]],
                                        [[-20.2785,237.803,4.09325],[0.991764,0.00796302,0.127826,-0.00113943],[-1,2,-1,1],[6093.43,9E+09,9E+09,9E+09,9E+09,9E+09]],
                                        [[-20.2723,238.832,4.10988],[0.991922,0.00899822,0.126523,-0.00112426],[-1,2,-1,1],[6095.43,9E+09,9E+09,9E+09,9E+09,9E+09]],
                                        [[-20.2663,239.865,4.12907],[0.992078,0.0100259,0.12522,-0.00110845],[-1,2,-1,1],[6097.43,9E+09,9E+09,9E+09,9E+09,9E+09]],
                                        [[-20.2612,240.892,4.14957],[0.99223,0.0110524,0.123917,-0.00108797],[-1,2,-1,1],[6099.43,9E+09,9E+09,9E+09,9E+09,9E+09]],
                                        [[-20.257,241.919,4.17177],[0.99238,0.0120803,0.122613,-0.00106264],[-1,2,-1,1],[6101.43,9E+09,9E+09,9E+09,9E+09,9E+09]],
                                        [[-20.2506,242.951,4.1963],[0.992528,0.013114,0.121308,-0.0010294],[-1,2,-1,1],[6103.43,9E+09,9E+09,9E+09,9E+09,9E+09]],
                                        [[-20.2442,243.991,4.22307],[0.992672,0.0141406,0.120004,-0.000983029],[-1,2,-1,1],[6105.43,9E+09,9E+09,9E+09,9E+09,9E+09]],
                                        [[-20.2401,245.027,4.25192],[0.992814,0.0151511,0.118699,-0.000933136],[-1,2,-1,1],[6107.43,9E+09,9E+09,9E+09,9E+09,9E+09]],
                                        [[-20.2344,246.071,4.27855],[0.992954,0.0161504,0.117394,-0.000885925],[-1,2,-1,1],[6109.43,9E+09,9E+09,9E+09,9E+09,9E+09]],
                                        [[-20.2256,247.114,4.31348],[0.99309,0.017147,0.116089,-0.000840642],[-1,2,-1,1],[6111.43,9E+09,9E+09,9E+09,9E+09,9E+09]],
                                        [[-20.2186,248.145,4.35501],[0.993225,0.018134,0.114783,-0.000805409],[-1,2,-1,1],[6113.43,9E+09,9E+09,9E+09,9E+09,9E+09]],
                                        [[-20.2127,249.175,4.39715],[0.993356,0.019121,0.113477,-0.000777209],[-1,2,-1,1],[6115.43,9E+09,9E+09,9E+09,9E+09,9E+09]],
                                        [[-20.2067,250.211,4.44015],[0.993485,0.0201063,0.11217,-0.000774825],[-1,2,-1,1],[6117.43,9E+09,9E+09,9E+09,9E+09,9E+09]],
                                        [[-20.2016,251.246,4.48539],[0.993612,0.0210878,0.110862,-0.000782539],[-1,2,-1,1],[6119.43,9E+09,9E+09,9E+09,9E+09,9E+09]],
                                        [[-20.1982,252.284,4.52948],[0.993735,0.0220742,0.109554,-0.000790505],[-1,2,-1,1],[6121.43,9E+09,9E+09,9E+09,9E+09,9E+09]],
                                        [[-20.1944,253.325,4.57549],[0.993856,0.0230695,0.108246,-0.00079446],[-1,2,-1,1],[6123.43,9E+09,9E+09,9E+09,9E+09,9E+09]],
                                        [[-20.1882,254.365,4.62621],[0.993974,0.0240811,0.106937,-0.000791414],[-1,2,-1,1],[6125.43,9E+09,9E+09,9E+09,9E+09,9E+09]],
                                        [[-20.1819,255.41,4.67734],[0.994089,0.0250925,0.105628,-0.000795986],[-1,2,-1,1],[6127.43,9E+09,9E+09,9E+09,9E+09,9E+09]],
                                        [[-20.1717,256.455,4.72485],[0.9942,0.0261308,0.104318,-0.000808304],[-1,2,-1,1],[6129.43,9E+09,9E+09,9E+09,9E+09,9E+09]],
                                        [[-20.1613,257.5,4.77974],[0.994309,0.0271881,0.103007,-0.00082828],[-1,2,-1,1],[6131.43,9E+09,9E+09,9E+09,9E+09,9E+09]],
                                        [[-20.1529,258.544,4.8362],[0.994414,0.0282578,0.101696,-0.00084936],[-1,2,-1,1],[6133.43,9E+09,9E+09,9E+09,9E+09,9E+09]],
                                        [[-20.1478,259.589,4.89401],[0.994383,0.029339,0.101686,-0.000833693],[-1,2,-1,1],[6135.43,9E+09,9E+09,9E+09,9E+09,9E+09]],
                                        [[-20.1415,260.639,4.95565],[0.994484,0.0304394,0.100375,-0.000833724],[-1,2,-1,1],[6137.43,9E+09,9E+09,9E+09,9E+09,9E+09]],
                                        [[-20.1357,261.692,5.01924],[0.994581,0.031543,0.0990631,-0.00082768],[-1,2,-1,1],[6139.43,9E+09,9E+09,9E+09,9E+09,9E+09]],
                                        [[-20.1295,262.746,5.083],[0.994675,0.032651,0.0977514,-0.000818514],[-1,2,-1,1],[6141.43,9E+09,9E+09,9E+09,9E+09,9E+09]],
                                        [[-20.1217,263.799,5.14856],[0.994766,0.0337691,0.0964394,-0.000805439],[-1,2,-1,1],[6143.43,9E+09,9E+09,9E+09,9E+09,9E+09]],
                                        [[-20.1134,264.861,5.21704],[0.994853,0.034892,0.0951271,-0.000796431],[-1,2,-1,1],[6145.43,9E+09,9E+09,9E+09,9E+09,9E+09]],
                                        [[-20.1048,265.922,5.28712],[0.994937,0.0360341,0.0938145,-0.000784898],[-1,2,-1,1],[6147.43,9E+09,9E+09,9E+09,9E+09,9E+09]],
                                        [[-20.0931,266.986,5.3615],[0.995017,0.0372133,0.0925016,-0.00076224],[-1,2,-1,1],[6149.43,9E+09,9E+09,9E+09,9E+09,9E+09]],
                                        [[-20.0749,268.043,5.4397],[0.995092,0.0384148,0.0911888,-0.000728855],[-1,2,-1,1],[6151.43,9E+09,9E+09,9E+09,9E+09,9E+09]],
                                        [[-20.0642,269.099,5.51988],[0.995164,0.0396363,0.0898762,-0.000680749],[-1,2,-1,1],[6153.43,9E+09,9E+09,9E+09,9E+09,9E+09]],
                                        [[-20.055,270.162,5.60375],[0.995231,0.0408896,0.0885636,-0.000619888],[-1,2,-1,1],[6155.43,9E+09,9E+09,9E+09,9E+09,9E+09]],
                                        [[-20.0452,271.226,5.69117],[0.995295,0.042134,0.0872516,-0.000550089],[-1,2,-1,1],[6157.43,9E+09,9E+09,9E+09,9E+09,9E+09]],
                                        [[-20.0359,272.285,5.7838],[0.995354,0.0433993,0.0859403,-0.000456421],[-1,2,-1,1],[6159.43,9E+09,9E+09,9E+09,9E+09,9E+09]],
                                        [[-20.0238,273.346,5.87181],[0.995298,0.0446997,0.0859318,-0.000299826],[-1,2,-1,1],[6161.43,9E+09,9E+09,9E+09,9E+09,9E+09]],
                                        [[-20.0121,274.414,5.9705],[0.995238,0.0460161,0.0859233,-0.000139029],[-1,2,-1,1],[6163.43,9E+09,9E+09,9E+09,9E+09,9E+09]],
                                        [[-19.9999,275.476,6.0724],[0.995177,0.0473426,0.0859147,2.33944E-05],[-1,2,-1,1],[6165.43,9E+09,9E+09,9E+09,9E+09,9E+09]],
                                        [[-19.9904,276.544,6.1745],[0.995114,0.048673,0.0859055,0.000175136],[-1,2,-1,1],[6167.43,9E+09,9E+09,9E+09,9E+09,9E+09]],
                                        [[-19.9793,277.608,6.27876],[0.995047,0.0500299,0.0858963,0.000333953],[-1,2,-1,1],[6169.43,9E+09,9E+09,9E+09,9E+09,9E+09]],
                                        [[-19.9769,278.672,6.39083],[0.994978,0.0513904,0.0858874,0.000500182],[-1,2,-1,1],[6171.43,9E+09,9E+09,9E+09,9E+09,9E+09]],
                                        [[-19.9711,279.738,6.49822],[0.994907,0.0527632,0.0858784,0.000669411],[-1,2,-1,1],[6169.43,9E+09,9E+09,9E+09,9E+09,9E+09]],
                                        [[-19.9636,280.805,6.60898],[0.994834,0.0541431,0.0858697,0.000846399],[-1,2,-1,1],[6171.43,9E+09,9E+09,9E+09,9E+09,9E+09]],
                                        [[-19.954,281.872,6.72454],[0.994758,0.0555176,0.0858619,0.00103767],[-1,2,-1,1],[6169.43,9E+09,9E+09,9E+09,9E+09,9E+09]],
                                        [[-19.9425,282.935,6.84487],[0.994682,0.056881,0.0858541,0.00122653],[-1,2,-1,1],[6171.43,9E+09,9E+09,9E+09,9E+09,9E+09]],
                                        [[-19.9361,284.003,6.96915],[0.994603,0.0582471,0.0858465,0.00141942],[-1,2,-1,1],[6173.43,9E+09,9E+09,9E+09,9E+09,9E+09]],
                                        [[-19.9313,285.072,7.09907],[0.994524,0.059597,0.0858393,0.00161381],[-1,2,-1,1],[6171.43,9E+09,9E+09,9E+09,9E+09,9E+09]],
                                        [[-19.926,286.141,7.22644],[0.994443,0.0609298,0.0858319,0.00180076],[-1,2,-1,1],[6173.43,9E+09,9E+09,9E+09,9E+09,9E+09]],
                                        [[-19.9226,287.204,7.35713],[0.994362,0.0622525,0.0858236,0.00196996],[-1,2,-1,1],[6171.43,9E+09,9E+09,9E+09,9E+09,9E+09]],
                                        [[-19.9172,288.267,7.49514],[0.994279,0.0635679,0.0858142,0.00212047],[-1,2,-1,1],[6173.43,9E+09,9E+09,9E+09,9E+09,9E+09]],
                                        [[-19.91,289.345,7.62309],[0.994195,0.0648717,0.0858043,0.00226003],[-1,2,-1,1],[6171.43,9E+09,9E+09,9E+09,9E+09,9E+09]],
                                        [[-19.908,290.444,7.76972],[0.994111,0.0661669,0.0857937,0.00238875],[-1,2,-1,1],[6173.43,9E+09,9E+09,9E+09,9E+09,9E+09]],
                                        [[-19.8998,291.548,7.92272],[0.994023,0.0674765,0.0857818,0.00250328],[-1,2,-1,1],[6175.43,9E+09,9E+09,9E+09,9E+09,9E+09]],
                                        [[-19.8907,292.644,8.07267],[0.993936,0.0687651,0.0857689,0.00260066],[-1,2,-1,1],[6173.43,9E+09,9E+09,9E+09,9E+09,9E+09]],
                                        [[-19.8845,293.743,8.22965],[0.993845,0.0700754,0.0857549,0.00268922],[-1,2,-1,1],[6175.43,9E+09,9E+09,9E+09,9E+09,9E+09]],
                                        [[-19.8737,294.843,8.38217],[0.993753,0.0713848,0.0857396,0.00276192],[-1,2,-1,1],[6173.43,9E+09,9E+09,9E+09,9E+09,9E+09]],
                                        [[-19.8678,295.949,8.54988],[0.993661,0.0726715,0.0857238,0.00282658],[-1,2,-1,1],[6175.43,9E+09,9E+09,9E+09,9E+09,9E+09]],
                                        [[-19.8596,297.049,8.71111],[0.993569,0.07394,0.0857074,0.00288316],[-1,2,-1,1],[6177.43,9E+09,9E+09,9E+09,9E+09,9E+09]],
                                        [[-19.85,298.155,8.87987],[0.993476,0.0751896,0.0856914,0.00294385],[-1,2,-1,1],[6175.43,9E+09,9E+09,9E+09,9E+09,9E+09]],
                                        [[-19.8422,299.253,9.04976],[0.993384,0.0764097,0.0856764,0.00301441],[-1,2,-1,1],[6177.43,9E+09,9E+09,9E+09,9E+09,9E+09]],
                                        [[-19.8385,300.353,9.22016],[0.993293,0.0775998,0.0856613,0.00308092],[-1,2,-1,1],[6175.43,9E+09,9E+09,9E+09,9E+09,9E+09]],
                                        [[-19.8287,301.452,9.39126],[0.9932,0.0787951,0.0856454,0.00314016],[-1,2,-1,1],[6177.43,9E+09,9E+09,9E+09,9E+09,9E+09]],
                                        [[-19.8221,302.552,9.57305],[0.993109,0.0799448,0.0856295,0.0031925],[-1,2,-1,1],[6175.43,9E+09,9E+09,9E+09,9E+09,9E+09]],
                                        [[-19.8155,303.65,9.75045],[0.99302,0.0810602,0.0856139,0.00324379],[-1,2,-1,1],[6177.43,9E+09,9E+09,9E+09,9E+09,9E+09]],
                                        [[-19.8083,304.749,9.92923],[0.992931,0.0821599,0.0855978,0.00328747],[-1,2,-1,1],[6175.43,9E+09,9E+09,9E+09,9E+09,9E+09]],
                                        [[-19.8031,305.848,10.1115],[0.992843,0.0832268,0.0855817,0.00332741],[-1,2,-1,1],[6177.43,9E+09,9E+09,9E+09,9E+09,9E+09]],
                                        [[-19.7905,306.94,10.2976],[0.992758,0.0842591,0.0855658,0.00336464],[-1,2,-1,1],[6179.43,9E+09,9E+09,9E+09,9E+09,9E+09]],
                                        [[-19.7799,308.032,10.4852],[0.992671,0.0852937,0.0855492,0.00339577],[-1,2,-1,1],[6177.43,9E+09,9E+09,9E+09,9E+09,9E+09]],
                                        [[-19.7694,309.123,10.6767],[0.992585,0.0862965,0.0855316,0.00341068],[-1,2,-1,1],[6179.43,9E+09,9E+09,9E+09,9E+09,9E+09]],
                                        [[-19.756,310.221,10.878],[0.9925,0.0872942,0.0855142,0.0034303],[-1,2,-1,1],[6177.43,9E+09,9E+09,9E+09,9E+09,9E+09]],
                                        [[-19.7455,311.32,11.0751],[0.992413,0.0882876,0.0854968,0.00345101],[-1,2,-1,1],[6179.43,9E+09,9E+09,9E+09,9E+09,9E+09]],
                                        [[-19.7367,312.402,11.2855],[0.992327,0.089268,0.085479,0.00346647],[-1,2,-1,1],[6177.43,9E+09,9E+09,9E+09,9E+09,9E+09]],
                                        [[-19.7266,313.462,11.4835],[0.992239,0.0902596,0.0854605,0.00347981],[-1,2,-1,1],[6179.43,9E+09,9E+09,9E+09,9E+09,9E+09]],
                                        [[-19.7183,314.519,11.678],[0.992152,0.0912296,0.0854419,0.00348889],[-1,2,-1,1],[6177.43,9E+09,9E+09,9E+09,9E+09,9E+09]],
                                        [[-19.7112,315.574,11.8757],[0.992061,0.0922289,0.0854233,0.00350744],[-1,2,-1,1],[6179.43,9E+09,9E+09,9E+09,9E+09,9E+09]],
                                        [[-19.7009,316.633,12.0713],[0.991971,0.0932061,0.0854052,0.00352854],[-1,2,-1,1],[6177.43,9E+09,9E+09,9E+09,9E+09,9E+09]],
                                        [[-19.6968,317.69,12.2725],[0.991883,0.0941535,0.0853886,0.0035617],[-1,2,-1,1],[6179.43,9E+09,9E+09,9E+09,9E+09,9E+09]],
                                        [[-19.6884,318.735,12.4713],[0.991795,0.0950812,0.085373,0.00360269],[-1,2,-1,1],[6177.43,9E+09,9E+09,9E+09,9E+09,9E+09]],
                                        [[-19.6793,319.768,12.6855],[0.99171,0.0959794,0.0853593,0.00365886],[-1,2,-1,1],[6179.43,9E+09,9E+09,9E+09,9E+09,9E+09]],
                                        [[-19.6745,320.793,12.8742],[0.991623,0.0968796,0.0853464,0.00372557],[-1,2,-1,1],[6177.43,9E+09,9E+09,9E+09,9E+09,9E+09]],
                                        [[-19.6671,321.825,13.0711],[0.991538,0.0977581,0.0853344,0.00379676],[-1,2,-1,1],[6179.43,9E+09,9E+09,9E+09,9E+09,9E+09]],
                                        [[-19.6538,322.862,13.2739],[0.991452,0.0986335,0.0853244,0.00388833],[-1,2,-1,1],[6177.43,9E+09,9E+09,9E+09,9E+09,9E+09]],
                                        [[-19.6434,323.901,13.4772],[0.991371,0.0994462,0.0853162,0.00398551],[-1,2,-1,1],[6179.43,9E+09,9E+09,9E+09,9E+09,9E+09]],
                                        [[-19.6307,324.95,13.6809],[0.991287,0.100278,0.0853092,0.00409867],[-1,2,-1,1],[6177.43,9E+09,9E+09,9E+09,9E+09,9E+09]],
                                        [[-19.6169,325.999,13.8984],[0.991198,0.101154,0.0853016,0.00421617],[-1,2,-1,1],[6179.43,9E+09,9E+09,9E+09,9E+09,9E+09]],
                                        [[-19.6009,327.052,14.1189],[0.99111,0.102014,0.0852943,0.00433272],[-1,2,-1,1],[6177.43,9E+09,9E+09,9E+09,9E+09,9E+09]],
                                        [[-19.5875,328.106,14.341],[0.991019,0.102899,0.0852878,0.00446199],[-1,2,-1,1],[6179.43,9E+09,9E+09,9E+09,9E+09,9E+09]],
                                        [[-19.5781,329.16,14.5634],[0.990923,0.10381,0.0852818,0.00460248],[-1,2,-1,1],[6177.43,9E+09,9E+09,9E+09,9E+09,9E+09]],
                                        [[-19.567,330.213,14.7877],[0.990826,0.104732,0.0852773,0.00475879],[-1,2,-1,1],[6179.43,9E+09,9E+09,9E+09,9E+09,9E+09]],
                                        [[-19.5529,331.26,15.0199],[0.990723,0.105699,0.0852744,0.00493892],[-1,2,-1,1],[6177.43,9E+09,9E+09,9E+09,9E+09,9E+09]],
                                        [[-19.5444,332.296,15.2454],[0.990617,0.106681,0.0852723,0.0051296],[-1,2,-1,1],[6179.43,9E+09,9E+09,9E+09,9E+09,9E+09]],
                                        [[-19.5344,333.319,15.4821],[0.990508,0.10768,0.0852711,0.00533133],[-1,2,-1,1],[6177.43,9E+09,9E+09,9E+09,9E+09,9E+09]],
                                        [[-19.5259,334.328,15.7024],[0.9904,0.108656,0.085271,0.00553715],[-1,2,-1,1],[6179.43,9E+09,9E+09,9E+09,9E+09,9E+09]],
                                        [[-19.5232,335.343,15.9187],[0.990293,0.109616,0.0852735,0.00576118],[-1,2,-1,1],[6177.43,9E+09,9E+09,9E+09,9E+09,9E+09]],
                                        [[-19.5166,336.363,16.1415],[0.990186,0.110559,0.0852787,0.00600571],[-1,2,-1,1],[6179.43,9E+09,9E+09,9E+09,9E+09,9E+09]],
                                        [[-19.5091,337.394,16.3668],[0.990081,0.11148,0.085285,0.00625226],[-1,2,-1,1],[6177.43,9E+09,9E+09,9E+09,9E+09,9E+09]],
                                        [[-19.5046,338.419,16.6067],[0.989968,0.112458,0.0852918,0.00651407],[-1,2,-1,1],[6179.43,9E+09,9E+09,9E+09,9E+09,9E+09]],
                                        [[-19.4954,339.448,16.8315],[0.989855,0.113422,0.0852993,0.00677587],[-1,2,-1,1],[6177.43,9E+09,9E+09,9E+09,9E+09,9E+09]],
                                        [[-19.492,340.476,17.0726],[0.989743,0.114379,0.0853077,0.00704215],[-1,2,-1,1],[6179.43,9E+09,9E+09,9E+09,9E+09,9E+09]],
                                        [[-19.4849,341.514,17.2912],[0.989629,0.115333,0.085315,0.00729667],[-1,2,-1,1],[6177.43,9E+09,9E+09,9E+09,9E+09,9E+09]],
                                        [[-19.4773,342.555,17.5485],[0.989518,0.116269,0.085321,0.00753285],[-1,2,-1,1],[6179.43,9E+09,9E+09,9E+09,9E+09,9E+09]],
                                        [[-19.4716,343.583,17.812],[0.989403,0.117226,0.0853255,0.00775917],[-1,2,-1,1],[6177.43,9E+09,9E+09,9E+09,9E+09,9E+09]],
                                        [[-19.4639,344.601,18.0521],[0.989287,0.118183,0.085327,0.00795806],[-1,2,-1,1],[6179.43,9E+09,9E+09,9E+09,9E+09,9E+09]],
                                        [[-19.4609,345.618,18.3099],[0.989165,0.119188,0.085325,0.00813603],[-1,2,-1,1],[6177.43,9E+09,9E+09,9E+09,9E+09,9E+09]],
                                        [[-19.4604,346.63,18.5619],[0.989043,0.120186,0.0853212,0.00829652],[-1,2,-1,1],[6179.43,9E+09,9E+09,9E+09,9E+09,9E+09]],
                                        [[-19.4603,347.633,18.8161],[0.988922,0.121171,0.085316,0.00844199],[-1,2,-1,1],[6177.43,9E+09,9E+09,9E+09,9E+09,9E+09]],
                                        [[-19.4614,348.641,19.0733],[0.988798,0.122177,0.0853093,0.00857954],[-1,2,-1,1],[6179.43,9E+09,9E+09,9E+09,9E+09,9E+09]],
                                        [[-19.4599,349.639,19.3255],[0.988677,0.123154,0.0852988,0.00867954],[-1,2,-1,1],[6177.43,9E+09,9E+09,9E+09,9E+09,9E+09]],
                                        [[-19.4572,350.631,19.5857],[0.988554,0.12414,0.0852855,0.00875971],[-1,2,-1,1],[6179.43,9E+09,9E+09,9E+09,9E+09,9E+09]],
                                        [[-19.4522,351.622,19.826],[0.988427,0.125153,0.0852703,0.00883031],[-1,2,-1,1],[6177.43,9E+09,9E+09,9E+09,9E+09,9E+09]],
                                        [[-19.4559,352.62,20.0793],[0.988302,0.126146,0.0852524,0.00887688],[-1,2,-1,1],[6179.43,9E+09,9E+09,9E+09,9E+09,9E+09]],
                                        [[-19.4552,353.633,20.3335],[0.988176,0.127134,0.0852353,0.0089301],[-1,2,-1,1],[6177.43,9E+09,9E+09,9E+09,9E+09,9E+09]],
                                        [[-19.4514,354.653,20.5879],[0.988053,0.128095,0.085218,0.00897718],[-1,2,-1,1],[6179.43,9E+09,9E+09,9E+09,9E+09,9E+09]],
                                        [[-19.4512,355.685,20.8683],[0.987928,0.129064,0.0851999,0.00902161],[-1,2,-1,1],[6177.43,9E+09,9E+09,9E+09,9E+09,9E+09]],
                                        [[-19.4431,356.706,21.142],[0.9878,0.130054,0.0851804,0.00905973],[-1,2,-1,1],[6179.43,9E+09,9E+09,9E+09,9E+09,9E+09]],
                                        [[-19.4396,357.729,21.4158],[0.987672,0.131036,0.0851576,0.00907311],[-1,2,-1,1],[6177.43,9E+09,9E+09,9E+09,9E+09,9E+09]],
                                        [[-19.4352,358.739,21.6893],[0.987542,0.132025,0.0851344,0.00908606],[-1,2,-1,1],[6179.43,9E+09,9E+09,9E+09,9E+09,9E+09]],
                                        [[-19.4257,359.759,21.9615],[0.98742,0.132951,0.0851098,0.00907826],[-1,2,-1,1],[6177.43,9E+09,9E+09,9E+09,9E+09,9E+09]],
                                        [[-19.4214,360.774,22.2574],[0.987293,0.133911,0.0850822,0.00905612],[-1,2,-1,1],[6179.43,9E+09,9E+09,9E+09,9E+09,9E+09]],
                                        [[-19.4115,361.793,22.5351],[0.987158,0.134921,0.0850533,0.00903644],[-1,2,-1,1],[6177.43,9E+09,9E+09,9E+09,9E+09,9E+09]],
                                        [[-19.4056,362.804,22.8356],[0.987022,0.135937,0.0850212,0.00899669],[-1,2,-1,1],[6179.43,9E+09,9E+09,9E+09,9E+09,9E+09]],
                                        [[-19.4006,363.829,23.1191],[0.986879,0.136992,0.0849899,0.00897308],[-1,2,-1,1],[6181.43,9E+09,9E+09,9E+09,9E+09,9E+09]],
                                        [[-19.3937,364.85,23.4022],[0.986733,0.138057,0.0849582,0.00895078],[-1,2,-1,1],[6179.43,9E+09,9E+09,9E+09,9E+09,9E+09]],
                                        [[-19.39,365.873,23.7015],[0.986583,0.139143,0.0849277,0.00894356],[-1,2,-1,1],[6181.43,9E+09,9E+09,9E+09,9E+09,9E+09]],
                                        [[-19.3794,366.895,23.9753],[0.986433,0.140225,0.0848979,0.00894355],[-1,2,-1,1],[6179.43,9E+09,9E+09,9E+09,9E+09,9E+09]],
                                        [[-19.3693,367.903,24.2692],[0.986279,0.141322,0.0848675,0.00894409],[-1,2,-1,1],[6181.43,9E+09,9E+09,9E+09,9E+09,9E+09]],
                                        [[-19.3646,368.931,24.5656],[0.986123,0.142423,0.0848368,0.0089456],[-1,2,-1,1],[6179.43,9E+09,9E+09,9E+09,9E+09,9E+09]],
                                        [[-19.354,369.946,24.8543],[0.985968,0.143509,0.0848067,0.00895069],[-1,2,-1,1],[6181.43,9E+09,9E+09,9E+09,9E+09,9E+09]],
                                        [[-19.3498,370.974,25.1635],[0.985808,0.144621,0.0847793,0.00898176],[-1,2,-1,1],[6183.43,9E+09,9E+09,9E+09,9E+09,9E+09]],
                                        [[-19.3447,372.002,25.4628],[0.98565,0.145701,0.0847554,0.00903221],[-1,2,-1,1],[6181.43,9E+09,9E+09,9E+09,9E+09,9E+09]],
                                        [[-19.3412,373.039,25.7853],[0.985497,0.146746,0.0847312,0.00907462],[-1,2,-1,1],[6183.43,9E+09,9E+09,9E+09,9E+09,9E+09]],
                                        [[-19.3323,374.076,26.1016],[0.985337,0.147819,0.0847109,0.00915125],[-1,2,-1,1],[6181.43,9E+09,9E+09,9E+09,9E+09,9E+09]],
                                        [[-19.3217,375.1,26.4225],[0.98518,0.148872,0.0846896,0.00921752],[-1,2,-1,1],[6183.43,9E+09,9E+09,9E+09,9E+09,9E+09]],
                                        [[-19.3146,376.134,26.7427],[0.985023,0.149915,0.0846695,0.00929133],[-1,2,-1,1],[6181.43,9E+09,9E+09,9E+09,9E+09,9E+09]],
                                        [[-19.3047,377.162,27.0589],[0.984866,0.150948,0.0846496,0.00936457],[-1,2,-1,1],[6183.43,9E+09,9E+09,9E+09,9E+09,9E+09]],
                                        [[-19.2945,378.205,27.3902],[0.984714,0.151943,0.0846292,0.00942821],[-1,2,-1,1],[6181.43,9E+09,9E+09,9E+09,9E+09,9E+09]],
                                        [[-19.2889,379.228,27.7184],[0.984558,0.152961,0.0846091,0.00949961],[-1,2,-1,1],[6183.43,9E+09,9E+09,9E+09,9E+09,9E+09]],
                                        [[-19.2771,380.259,28.0552],[0.984405,0.153951,0.0845881,0.00956022],[-1,2,-1,1],[6181.43,9E+09,9E+09,9E+09,9E+09,9E+09]],
                                        [[-19.2747,381.273,28.3874],[0.984246,0.154968,0.0845671,0.00962728],[-1,2,-1,1],[6183.43,9E+09,9E+09,9E+09,9E+09,9E+09]],
                                        [[-19.2646,382.294,28.7178],[0.98409,0.155963,0.0845482,0.00970385],[-1,2,-1,1],[6181.43,9E+09,9E+09,9E+09,9E+09,9E+09]],
                                        [[-19.2588,383.307,29.0523],[0.983937,0.156935,0.0845278,0.00976707],[-1,2,-1,1],[6183.43,9E+09,9E+09,9E+09,9E+09,9E+09]],
                                        [[-19.2491,384.34,29.3833],[0.983781,0.15791,0.0845095,0.00984551],[-1,2,-1,1],[6181.43,9E+09,9E+09,9E+09,9E+09,9E+09]],
                                        [[-19.2378,385.352,29.7215],[0.983635,0.158828,0.0844889,0.00989836],[-1,2,-1,1],[6183.43,9E+09,9E+09,9E+09,9E+09,9E+09]],
                                        [[-19.228,386.378,30.0535],[0.983488,0.159741,0.0844671,0.00994322],[-1,2,-1,1],[6181.43,9E+09,9E+09,9E+09,9E+09,9E+09]],
                                        [[-19.2222,387.403,30.4007],[0.983345,0.160628,0.0844461,0.00998939],[-1,2,-1,1],[6183.43,9E+09,9E+09,9E+09,9E+09,9E+09]],
                                        [[-19.2151,388.426,30.76],[0.983205,0.16149,0.0844258,0.0100357],[-1,2,-1,1],[6185.43,9E+09,9E+09,9E+09,9E+09,9E+09]],
                                        [[-19.2114,389.453,31.1058],[0.983066,0.162342,0.0844076,0.010093],[-1,2,-1,1],[6183.43,9E+09,9E+09,9E+09,9E+09,9E+09]],
                                        [[-19.1989,390.466,31.4495],[0.982929,0.163173,0.0843914,0.0101591],[-1,2,-1,1],[6185.43,9E+09,9E+09,9E+09,9E+09,9E+09]],
                                        [[-19.1981,391.484,31.8077],[0.98279,0.164014,0.0843752,0.0102282],[-1,2,-1,1],[6183.43,9E+09,9E+09,9E+09,9E+09,9E+09]],
                                        [[-19.1881,392.489,32.1462],[0.982648,0.164863,0.0843587,0.0102974],[-1,2,-1,1],[6185.43,9E+09,9E+09,9E+09,9E+09,9E+09]],
                                        [[-19.1806,393.5,32.4965],[0.982501,0.165745,0.0843393,0.0103557],[-1,2,-1,1],[6183.43,9E+09,9E+09,9E+09,9E+09,9E+09]],
                                        [[-19.1701,394.499,32.8442],[0.98235,0.166646,0.0843196,0.0104171],[-1,2,-1,1],[6185.43,9E+09,9E+09,9E+09,9E+09,9E+09]],
                                        [[-19.1624,395.497,33.1858],[0.982197,0.167551,0.0842971,0.0104625],[-1,2,-1,1],[6183.43,9E+09,9E+09,9E+09,9E+09,9E+09]],
                                        [[-19.154,396.493,33.5345],[0.982038,0.168494,0.0842719,0.0105011],[-1,2,-1,1],[6185.43,9E+09,9E+09,9E+09,9E+09,9E+09]],
                                        [[-19.1455,397.487,33.8818],[0.981874,0.169455,0.0842472,0.0105465],[-1,2,-1,1],[6183.43,9E+09,9E+09,9E+09,9E+09,9E+09]],
                                        [[-19.1381,398.492,34.2354],[0.981703,0.170451,0.0842195,0.0105831],[-1,2,-1,1],[6185.43,9E+09,9E+09,9E+09,9E+09,9E+09]],
                                        [[-19.1325,399.482,34.588],[0.981522,0.171501,0.084192,0.0106322],[-1,2,-1,1],[6183.43,9E+09,9E+09,9E+09,9E+09,9E+09]],
                                        [[-19.1196,400.478,34.9453],[0.981337,0.172572,0.0841637,0.0106819],[-1,2,-1,1],[6185.43,9E+09,9E+09,9E+09,9E+09,9E+09]],
                                        [[-19.1137,401.47,35.3035],[0.981141,0.173688,0.0841358,0.0107445],[-1,2,-1,1],[6183.43,9E+09,9E+09,9E+09,9E+09,9E+09]],
                                        [[-19.1001,402.47,35.6621],[0.980946,0.174798,0.0841068,0.0108001],[-1,2,-1,1],[6185.43,9E+09,9E+09,9E+09,9E+09,9E+09]],
                                        [[-19.0915,403.46,36.0229],[0.980739,0.175967,0.0840766,0.0108623],[-1,2,-1,1],[6183.43,9E+09,9E+09,9E+09,9E+09,9E+09]],
                                        [[-19.0817,404.457,36.3875],[0.980534,0.177119,0.0840437,0.0109073],[-1,2,-2,1],[6185.43,9E+09,9E+09,9E+09,9E+09,9E+09]],
                                        [[-19.0773,405.444,36.7542],[0.980326,0.178279,0.0840126,0.0109652],[-1,2,-2,1],[6183.43,9E+09,9E+09,9E+09,9E+09,9E+09]],
                                        [[-19.071,406.441,37.1212],[0.980113,0.179457,0.0839813,0.0110269],[-1,2,-2,1],[6185.43,9E+09,9E+09,9E+09,9E+09,9E+09]],
                                        [[-19.0643,407.428,37.4934],[0.979896,0.180644,0.0839531,0.011109],[-1,2,-2,1],[6187.43,9E+09,9E+09,9E+09,9E+09,9E+09]],
                                        [[-19.0525,408.41,37.8639],[0.979675,0.181845,0.0839241,0.0111899],[-1,2,-2,1],[6185.43,9E+09,9E+09,9E+09,9E+09,9E+09]],
                                        [[-19.0448,409.389,38.2394],[0.97945,0.183065,0.0838961,0.0112819],[-1,2,-2,1],[6187.43,9E+09,9E+09,9E+09,9E+09,9E+09]],
                                        [[-19.0333,410.375,38.6261],[0.979217,0.18431,0.0838687,0.0113825],[-1,2,-2,1],[6185.43,9E+09,9E+09,9E+09,9E+09,9E+09]],
                                        [[-19.0244,411.361,39.0165],[0.978985,0.185545,0.083839,0.01147],[-1,2,-2,1],[6187.43,9E+09,9E+09,9E+09,9E+09,9E+09]],
                                        [[-19.011,412.341,39.4036],[0.978751,0.186787,0.0838099,0.0115631],[-1,2,-2,1],[6185.43,9E+09,9E+09,9E+09,9E+09,9E+09]],
                                        [[-19.0001,413.328,39.8018],[0.978519,0.188002,0.0837809,0.011652],[-1,2,-2,1],[6187.43,9E+09,9E+09,9E+09,9E+09,9E+09]],
                                        [[-18.9908,414.312,40.1954],[0.978291,0.189192,0.083752,0.0117376],[-1,2,-2,1],[6185.43,9E+09,9E+09,9E+09,9E+09,9E+09]],
                                        [[-18.9808,415.297,40.5926],[0.978067,0.190357,0.0837253,0.0118304],[-1,2,-2,1],[6187.43,9E+09,9E+09,9E+09,9E+09,9E+09]],
                                        [[-18.9692,416.281,41.0024],[0.977846,0.191494,0.0837004,0.0119277],[-1,2,-2,1],[6185.43,9E+09,9E+09,9E+09,9E+09,9E+09]],
                                        [[-18.9614,417.264,41.406],[0.977628,0.192608,0.0836766,0.0120272],[-1,2,-2,1],[6187.43,9E+09,9E+09,9E+09,9E+09,9E+09]],
                                        [[-18.9537,418.24,41.8155],[0.977413,0.1937,0.0836497,0.0121063],[-1,2,-2,1],[6189.43,9E+09,9E+09,9E+09,9E+09,9E+09]],
                                        [[-18.9431,419.211,42.2177],[0.977199,0.194786,0.0836234,0.0121888],[-1,2,-2,1],[6187.43,9E+09,9E+09,9E+09,9E+09,9E+09]],
                                        [[-18.9379,420.179,42.6383],[0.976991,0.195835,0.0835935,0.0122459],[-1,2,-2,1],[6189.43,9E+09,9E+09,9E+09,9E+09,9E+09]],
                                        [[-18.9241,421.152,43.0395],[0.976786,0.196861,0.0835637,0.0122996],[-1,2,-2,1],[6187.43,9E+09,9E+09,9E+09,9E+09,9E+09]],
                                        [[-18.917,422.125,43.4449],[0.976587,0.197858,0.0835333,0.0123457],[-1,2,-2,1],[6189.43,9E+09,9E+09,9E+09,9E+09,9E+09]],
                                        [[-18.9077,423.099,43.8477],[0.976388,0.198845,0.0835039,0.0123956],[-1,2,-2,1],[6187.43,9E+09,9E+09,9E+09,9E+09,9E+09]],
                                        [[-18.9018,424.073,44.264],[0.976198,0.199787,0.083474,0.0124351],[-1,2,-2,1],[6189.43,9E+09,9E+09,9E+09,9E+09,9E+09]],
                                        [[-18.8955,425.045,44.6827],[0.976006,0.200734,0.0834456,0.0124835],[-1,2,-2,1],[6187.43,9E+09,9E+09,9E+09,9E+09,9E+09]],
                                        [[-18.8823,426.022,45.0994],[0.975813,0.201677,0.0834144,0.0125184],[-1,2,-2,1],[6189.43,9E+09,9E+09,9E+09,9E+09,9E+09]],
                                        [[-18.8771,426.984,45.5337],[0.975616,0.202642,0.0833827,0.0125558],[-1,2,-2,1],[6187.43,9E+09,9E+09,9E+09,9E+09,9E+09]],
                                        [[-18.8616,427.953,45.9499],[0.975426,0.203568,0.0833472,0.012568],[-1,2,-2,1],[6189.43,9E+09,9E+09,9E+09,9E+09,9E+09]],
                                        [[-18.8559,428.93,46.3794],[0.975235,0.204495,0.0833122,0.0125837],[-1,2,-2,1],[6187.43,9E+09,9E+09,9E+09,9E+09,9E+09]],
                                        [[-18.8446,429.908,46.8029],[0.975044,0.205415,0.0832754,0.0125903],[-1,2,-2,1],[6189.43,9E+09,9E+09,9E+09,9E+09,9E+09]],
                                        [[-18.8346,430.875,47.2254],[0.974859,0.206309,0.083236,0.0125801],[-1,2,-2,1],[6187.43,9E+09,9E+09,9E+09,9E+09,9E+09]],
                                        [[-18.8284,431.848,47.651],[0.974671,0.20721,0.0831973,0.0125765],[-1,2,-2,1],[6189.43,9E+09,9E+09,9E+09,9E+09,9E+09]],
                                        [[-18.8205,432.816,48.0763],[0.974487,0.208091,0.0831579,0.012566],[-1,2,-2,1],[6191.43,9E+09,9E+09,9E+09,9E+09,9E+09]],
                                        [[-18.8097,433.773,48.5027],[0.974297,0.208995,0.0831156,0.0125476],[-1,2,-2,1],[6189.43,9E+09,9E+09,9E+09,9E+09,9E+09]],
                                        [[-18.7965,434.736,48.9298],[0.974107,0.209898,0.0830747,0.0125367],[-1,2,-2,1],[6191.43,9E+09,9E+09,9E+09,9E+09,9E+09]],
                                        [[-18.7857,435.696,49.3697],[0.973916,0.210802,0.0830326,0.0125218],[-1,2,-2,1],[6189.43,9E+09,9E+09,9E+09,9E+09,9E+09]],
                                        [[-18.7714,436.66,49.8009],[0.973721,0.211717,0.0829897,0.0125068],[-1,2,-2,1],[6191.43,9E+09,9E+09,9E+09,9E+09,9E+09]],
                                        [[-18.7606,437.625,50.2418],[0.973519,0.212658,0.0829507,0.0125165],[-1,2,-2,1],[6189.43,9E+09,9E+09,9E+09,9E+09,9E+09]],
                                        [[-18.7492,438.596,50.6841],[0.973315,0.213606,0.0829097,0.0125188],[-1,2,-2,1],[6191.43,9E+09,9E+09,9E+09,9E+09,9E+09]],
                                        [[-18.7361,439.564,51.1352],[0.973111,0.214547,0.0828715,0.0125341],[-1,2,-2,1],[6189.43,9E+09,9E+09,9E+09,9E+09,9E+09]],
                                        [[-18.7199,440.535,51.5786],[0.9728,0.215455,0.0841087,0.0128383],[-1,2,-2,1],[6191.43,9E+09,9E+09,9E+09,9E+09,9E+09]],
                                        [[-18.71,441.505,52.0405],[0.972592,0.216403,0.0840736,0.0128735],[-1,2,-2,1],[6189.43,9E+09,9E+09,9E+09,9E+09,9E+09]],
                                        [[-18.696,442.475,52.5051],[0.972385,0.217344,0.0840401,0.0129154],[-1,2,-2,1],[6191.43,9E+09,9E+09,9E+09,9E+09,9E+09]],
                                        [[-18.6835,443.436,52.9777],[0.972174,0.218297,0.0840057,0.0129567],[-1,2,-2,1],[6189.43,9E+09,9E+09,9E+09,9E+09,9E+09]],
                                        [[-18.6653,444.404,53.4193],[0.971952,0.219293,0.0839725,0.0130131],[-1,2,-2,1],[6191.43,9E+09,9E+09,9E+09,9E+09,9E+09]],
                                        [[-18.6544,445.368,53.8787],[0.971726,0.2203,0.0839387,0.0130692],[-1,2,-2,1],[6189.43,9E+09,9E+09,9E+09,9E+09,9E+09]],
                                        [[-18.6432,446.334,54.3396],[0.971498,0.22131,0.0839059,0.0131321],[-1,2,-2,1],[6191.43,9E+09,9E+09,9E+09,9E+09,9E+09]],
                                        [[-18.627,447.301,54.7911],[0.971276,0.222291,0.0838766,0.0132046],[-1,2,-2,1],[6189.43,9E+09,9E+09,9E+09,9E+09,9E+09]],
                                        [[-18.6176,448.267,55.2635],[0.971051,0.223278,0.0838502,0.0132923],[-1,2,-2,1],[6191.43,9E+09,9E+09,9E+09,9E+09,9E+09]],
                                        [[-18.6039,449.233,55.7251],[0.970823,0.224269,0.0838254,0.0133881],[-1,2,-2,1],[6189.43,9E+09,9E+09,9E+09,9E+09,9E+09]],
                                        [[-18.5896,450.194,56.1976],[0.970596,0.22525,0.0838059,0.0135049],[-1,2,-2,1],[6191.43,9E+09,9E+09,9E+09,9E+09,9E+09]],
                                        [[-18.5787,451.16,56.667],[0.970366,0.226239,0.0837852,0.0136188],[-1,2,-2,1],[6193.43,9E+09,9E+09,9E+09,9E+09,9E+09]],
                                        [[-18.5627,452.12,57.1354],[0.970132,0.227241,0.0837651,0.0137381],[-1,2,-2,1],[6191.43,9E+09,9E+09,9E+09,9E+09,9E+09]],
                                        [[-18.5503,453.088,57.6143],[0.969779,0.228256,0.0850126,0.0141545],[-1,2,-2,1],[6189.43,9E+09,9E+09,9E+09,9E+09,9E+09]],
                                        [[-18.5419,454.068,58.0989],[0.969419,0.229291,0.0862589,0.0145765],[-1,2,-2,1],[6187.43,9E+09,9E+09,9E+09,9E+09,9E+09]],
                                        [[-18.5298,455.038,58.5873],[0.969052,0.230338,0.0875028,0.0149969],[-1,2,-2,1],[6185.43,9E+09,9E+09,9E+09,9E+09,9E+09]],
                                        [[-18.5198,456.006,59.0738],[0.968675,0.231417,0.0887463,0.0154294],[-1,2,-2,1],[6183.43,9E+09,9E+09,9E+09,9E+09,9E+09]],
                                        [[-18.5096,456.972,59.5624],[0.968294,0.232503,0.0899859,0.0158537],[-1,2,-2,1],[6181.43,9E+09,9E+09,9E+09,9E+09,9E+09]],
                                        [[-18.4967,457.93,60.0557],[0.967918,0.233559,0.0912207,0.0162582],[-1,2,-2,1],[6179.43,9E+09,9E+09,9E+09,9E+09,9E+09]],
                                        [[-18.4825,458.886,60.5365],[0.967536,0.234624,0.0924546,0.0166681],[-1,2,-2,1],[6177.43,9E+09,9E+09,9E+09,9E+09,9E+09]],
                                        [[-18.4716,459.836,61.0333],[0.967147,0.235706,0.0936866,0.0170801],[-1,2,-2,1],[6175.43,9E+09,9E+09,9E+09,9E+09,9E+09]],
                                        [[-18.4575,460.787,61.5221],[0.966746,0.236827,0.0949182,0.0175074],[-1,2,-2,1],[6173.43,9E+09,9E+09,9E+09,9E+09,9E+09]],
                                        [[-18.4495,461.73,62.0191],[0.966355,0.237893,0.0961465,0.0179156],[-1,2,-2,1],[6171.43,9E+09,9E+09,9E+09,9E+09,9E+09]],
                                        [[-18.4341,462.661,62.5058],[0.965959,0.238969,0.0973738,0.0183289],[-1,2,-2,1],[6169.43,9E+09,9E+09,9E+09,9E+09,9E+09]],
                                        [[-18.4261,463.61,62.9886],[0.965567,0.240014,0.0986027,0.0187489],[-1,2,-2,1],[6167.43,9E+09,9E+09,9E+09,9E+09,9E+09]],
                                        [[-18.4184,464.551,63.4933],[0.965184,0.241011,0.09983,0.0191579],[-1,2,-2,1],[6165.43,9E+09,9E+09,9E+09,9E+09,9E+09]],
                                        [[-18.4038,465.493,63.9931],[0.964932,0.242026,0.0997948,0.0192572],[-1,2,-2,1],[6163.44,9E+09,9E+09,9E+09,9E+09,9E+09]],
                                        [[-18.3966,466.429,64.4949],[0.964552,0.242997,0.101023,0.0196746],[-1,2,-2,1],[6161.47,9E+09,9E+09,9E+09,9E+09,9E+09]],
                                        [[-18.3817,467.376,65.0042],[0.964163,0.243994,0.102245,0.0200781],[-1,2,-2,1],[6159.55,9E+09,9E+09,9E+09,9E+09,9E+09]],
                                        [[-18.3726,468.312,65.5191],[0.963764,0.245022,0.103463,0.0204807],[-1,2,-2,1],[6157.65,9E+09,9E+09,9E+09,9E+09,9E+09]],
                                        [[-18.3573,469.247,66.0354],[0.963367,0.246033,0.104677,0.0208706],[-1,2,-2,1],[6155.78,9E+09,9E+09,9E+09,9E+09,9E+09]],
                                        [[-18.3484,470.18,66.5566],[0.962961,0.247065,0.105889,0.0212633],[-1,2,-2,1],[6153.96,9E+09,9E+09,9E+09,9E+09,9E+09]],
                                        [[-18.3325,471.11,67.0755],[0.96256,0.248069,0.107102,0.0216634],[-1,2,-2,1],[6152.16,9E+09,9E+09,9E+09,9E+09,9E+09]],
                                        [[-18.3222,472.032,67.6021],[0.962164,0.249041,0.108316,0.0220652],[-1,2,-2,1],[6150.38,9E+09,9E+09,9E+09,9E+09,9E+09]],
                                        [[-18.3065,472.953,68.1127],[0.961775,0.249973,0.10953,0.0224617],[-1,2,-2,1],[6148.64,9E+09,9E+09,9E+09,9E+09,9E+09]],
                                        [[-18.2903,473.872,68.6178],[0.961389,0.250885,0.110745,0.022865],[-1,2,-2,1],[6146.9,9E+09,9E+09,9E+09,9E+09,9E+09]],
                                        [[-18.2763,474.803,69.1344],[0.961001,0.251796,0.11196,0.0232752],[-1,2,-2,1],[6145.18,9E+09,9E+09,9E+09,9E+09,9E+09]],
                                        [[-18.2647,475.723,69.6515],[0.96062,0.252665,0.113174,0.0236772],[-1,2,-2,1],[6143.47,9E+09,9E+09,9E+09,9E+09,9E+09]],
                                        [[-18.2562,476.638,70.1683],[0.960234,0.253546,0.114389,0.0240918],[-1,2,-2,1],[6141.78,9E+09,9E+09,9E+09,9E+09,9E+09]],
                                        [[-18.2437,477.561,70.6808],[0.959992,0.254471,0.114346,0.0241777],[-1,2,-2,1],[6140.17,9E+09,9E+09,9E+09,9E+09,9E+09]],
                                        [[-18.231,478.489,71.2104],[0.959742,0.255421,0.114307,0.0242862],[-1,2,-2,1],[6138.62,9E+09,9E+09,9E+09,9E+09,9E+09]],
                                        [[-18.221,479.409,71.7249],[0.959501,0.256337,0.114264,0.0243672],[-1,2,-2,1],[6137.14,9E+09,9E+09,9E+09,9E+09,9E+09]],
                                        [[-18.2096,480.338,72.2501],[0.959271,0.257207,0.114221,0.0244424],[-1,2,-2,1],[6135.72,9E+09,9E+09,9E+09,9E+09,9E+09]],
                                        [[-18.197,481.269,72.7734],[0.959039,0.25808,0.114181,0.0245261],[-1,2,-2,1],[6134.36,9E+09,9E+09,9E+09,9E+09,9E+09]],
                                        [[-18.1873,482.199,73.3149],[0.958808,0.258947,0.11414,0.0246072],[-1,2,-2,1],[6133.05,9E+09,9E+09,9E+09,9E+09,9E+09]],
                                        [[-18.1702,483.115,73.8584],[0.958579,0.259802,0.114104,0.0247029],[-1,2,-2,1],[6131.8,9E+09,9E+09,9E+09,9E+09,9E+09]],
                                        [[-18.1545,484.024,74.4105],[0.958349,0.260653,0.114069,0.0248023],[-1,2,-2,1],[6130.62,9E+09,9E+09,9E+09,9E+09,9E+09]],
                                        [[-18.1409,484.942,74.9514],[0.957962,0.261496,0.115288,0.0252531],[-1,2,-2,1],[6129.49,9E+09,9E+09,9E+09,9E+09,9E+09]],
                                        [[-18.1284,485.846,75.5028],[0.957723,0.262374,0.115254,0.0253655],[-1,2,-2,1],[6128.39,9E+09,9E+09,9E+09,9E+09,9E+09]],
                                        [[-18.1154,486.747,76.0345],[0.957475,0.263278,0.115224,0.0255009],[-1,2,-2,1],[6130.39,9E+09,9E+09,9E+09,9E+09,9E+09]],
                                        [[-18.1041,487.655,76.5604],[0.957224,0.264189,0.115194,0.0256399],[-1,2,-2,1],[6129.26,9E+09,9E+09,9E+09,9E+09,9E+09]],
                                        [[-18.088,488.567,77.0938],[0.956957,0.265154,0.115163,0.02579],[-1,2,-2,1],[6128.17,9E+09,9E+09,9E+09,9E+09,9E+09]],
                                        [[-18.0762,489.478,77.6333],[0.956694,0.266102,0.115126,0.0259166],[-1,2,-2,1],[6130.17,9E+09,9E+09,9E+09,9E+09,9E+09]],
                                        [[-18.0659,490.385,78.1823],[0.956434,0.267038,0.115093,0.0260497],[-1,2,-2,1],[6129.04,9E+09,9E+09,9E+09,9E+09,9E+09]],
                                        [[-18.0532,491.296,78.7228],[0.956169,0.267987,0.115057,0.0261785],[-1,2,-2,1],[6127.97,9E+09,9E+09,9E+09,9E+09,9E+09]],
                                        [[-18.0431,492.196,79.2742],[0.9559,0.268943,0.115025,0.0263255],[-1,2,-2,1],[6129.97,9E+09,9E+09,9E+09,9E+09,9E+09]],
                                        [[-18.0328,493.096,79.8382],[0.955631,0.269894,0.114998,0.0264863],[-1,2,-2,1],[6128.86,9E+09,9E+09,9E+09,9E+09,9E+09]],
                                        [[-18.0245,493.976,80.3909],[0.955378,0.270785,0.114974,0.0266428],[-1,2,-2,1],[6127.79,9E+09,9E+09,9E+09,9E+09,9E+09]],
                                        [[-18.0068,494.87,80.9261],[0.955123,0.271676,0.11495,0.0267992],[-1,2,-2,1],[6129.79,9E+09,9E+09,9E+09,9E+09,9E+09]],
                                        [[-17.9902,495.755,81.4728],[0.954877,0.272532,0.114929,0.0269604],[-1,2,-2,1],[6128.66,9E+09,9E+09,9E+09,9E+09,9E+09]],
                                        [[-17.976,496.635,82.0175],[0.95449,0.273313,0.116162,0.0274792],[-1,2,-2,1],[6127.52,9E+09,9E+09,9E+09,9E+09,9E+09]],
                                        [[-17.9651,497.508,82.5661],[0.95412,0.274026,0.117396,0.0279906],[-1,2,-2,1],[6126.34,9E+09,9E+09,9E+09,9E+09,9E+09]],
                                        [[-17.9533,498.403,83.1205],[0.953742,0.274751,0.118636,0.0285321],[-1,2,-2,1],[6125.14,9E+09,9E+09,9E+09,9E+09,9E+09]],
                                        [[-17.9444,499.279,83.6767],[0.953357,0.275492,0.119873,0.0290745],[-1,2,-2,1],[6123.88,9E+09,9E+09,9E+09,9E+09,9E+09]],
                                        [[-17.9309,500.166,84.2395],[0.952957,0.276277,0.121107,0.0296216],[-1,2,-2,1],[6122.62,9E+09,9E+09,9E+09,9E+09,9E+09]],
                                        [[-17.922,501.053,84.8004],[0.952561,0.277036,0.122342,0.0301677],[-1,2,-2,1],[6121.32,9E+09,9E+09,9E+09,9E+09,9E+09]],
                                        [[-17.9134,501.944,85.3705],[0.952148,0.27785,0.123572,0.0307182],[-1,2,-2,1],[6119.99,9E+09,9E+09,9E+09,9E+09,9E+09]],
                                        [[-17.9055,502.839,85.9363],[0.951726,0.278686,0.124798,0.0312678],[-1,2,-2,1],[6118.64,9E+09,9E+09,9E+09,9E+09,9E+09]],
                                        [[-17.8934,503.72,86.5128],[0.951303,0.27951,0.126026,0.031829],[-1,2,-2,1],[6117.26,9E+09,9E+09,9E+09,9E+09,9E+09]],
                                        [[-17.8763,504.607,87.0714],[0.950882,0.280323,0.127252,0.0323816],[-1,2,-2,1],[6115.88,9E+09,9E+09,9E+09,9E+09,9E+09]],
                                        [[-17.8712,505.484,87.6433],[0.950462,0.281122,0.12848,0.0329412],[-1,2,-2,1],[6114.46,9E+09,9E+09,9E+09,9E+09,9E+09]],
                                        [[-17.8594,506.354,88.2177],[0.950042,0.281907,0.12971,0.0335124],[-1,2,-2,1],[6113.03,9E+09,9E+09,9E+09,9E+09,9E+09]],
                                        [[-17.854,507.217,88.785],[0.949634,0.282645,0.130943,0.0340843],[-1,2,-2,1],[6111.59,9E+09,9E+09,9E+09,9E+09,9E+09]],
                                        [[-17.8446,508.083,89.3462],[0.949221,0.283382,0.13218,0.0346754],[-1,2,-2,1],[6110.12,9E+09,9E+09,9E+09,9E+09,9E+09]],
                                        [[-17.8348,508.955,89.9046],[0.948798,0.284144,0.133415,0.0352717],[-1,2,-2,1],[6108.62,9E+09,9E+09,9E+09,9E+09,9E+09]],
                                        [[-17.8241,509.82,90.4724],[0.948365,0.284929,0.134653,0.0358885],[-1,2,-2,1],[6107.09,9E+09,9E+09,9E+09,9E+09,9E+09]],
                                        [[-17.8142,510.695,91.0452],[0.947933,0.2857,0.135888,0.0364984],[-1,2,-2,1],[6105.55,9E+09,9E+09,9E+09,9E+09,9E+09]],
                                        [[-17.8041,511.562,91.6079],[0.94767,0.286547,0.135878,0.0367291],[-1,2,-2,1],[6103.99,9E+09,9E+09,9E+09,9E+09,9E+09]],
                                        [[-17.7925,512.436,92.1743],[0.947229,0.287347,0.137103,0.0373206],[-1,2,-2,1],[6102.4,9E+09,9E+09,9E+09,9E+09,9E+09]],
                                        [[-17.7889,513.31,92.7655],[0.946775,0.288178,0.138325,0.0379166],[-1,2,-2,1],[6100.8,9E+09,9E+09,9E+09,9E+09,9E+09]],
                                        [[-17.7822,514.188,93.3507],[0.946306,0.289054,0.139538,0.0385022],[-1,2,-2,1],[6099.2,9E+09,9E+09,9E+09,9E+09,9E+09]],
                                        [[-17.7743,515.061,93.9442],[0.945817,0.289986,0.140746,0.0390982],[-1,2,-2,1],[6097.58,9E+09,9E+09,9E+09,9E+09,9E+09]],
                                        [[-17.7663,515.944,94.5244],[0.945312,0.290964,0.141947,0.0396889],[-1,2,-2,1],[6095.96,9E+09,9E+09,9E+09,9E+09,9E+09]],
                                        [[-17.7551,516.81,95.1237],[0.944794,0.291979,0.143144,0.040282],[-1,2,-2,1],[6094.33,9E+09,9E+09,9E+09,9E+09,9E+09]],
                                        [[-17.7447,517.681,95.7243],[0.944258,0.293042,0.144334,0.0408792],[-1,2,-2,1],[6092.73,9E+09,9E+09,9E+09,9E+09,9E+09]],
                                        [[-17.7389,518.536,96.3244],[0.943716,0.294111,0.145527,0.0414943],[-1,2,-2,1],[6091.12,9E+09,9E+09,9E+09,9E+09,9E+09]],
                                        [[-17.7308,519.39,96.9161],[0.943144,0.295263,0.146713,0.0421196],[-1,2,-2,1],[6089.52,9E+09,9E+09,9E+09,9E+09,9E+09]],
                                        [[-17.7247,520.235,97.4973],[0.942585,0.296372,0.147893,0.0427221],[-1,2,-2,1],[6087.93,9E+09,9E+09,9E+09,9E+09,9E+09]],
                                        [[-17.7192,521.083,98.0818],[0.942018,0.297491,0.149075,0.0433415],[-1,2,-2,1],[6086.35,9E+09,9E+09,9E+09,9E+09,9E+09]],
                                        [[-17.714,521.936,98.6617],[0.941448,0.29861,0.150252,0.0439485],[-1,2,-2,1],[6084.77,9E+09,9E+09,9E+09,9E+09,9E+09]],
                                        [[-17.7114,522.789,99.2555],[0.941067,0.299809,0.150192,0.0441665],[-1,2,-2,1],[6083.26,9E+09,9E+09,9E+09,9E+09,9E+09]],
                                        [[-17.7021,523.65,99.8556],[0.940689,0.300995,0.150127,0.0443611],[-1,2,-2,1],[6081.82,9E+09,9E+09,9E+09,9E+09,9E+09]],
                                        [[-17.697,524.516,100.464],[0.940118,0.302116,0.151285,0.0449239],[-1,2,-2,1],[6080.45,9E+09,9E+09,9E+09,9E+09,9E+09]],
                                        [[-17.6936,525.387,101.086],[0.939734,0.303325,0.151202,0.0450732],[-1,2,-2,1],[6079.15,9E+09,9E+09,9E+09,9E+09,9E+09]],
                                        [[-17.6886,526.251,101.707],[0.939355,0.304521,0.151114,0.0452039],[-1,2,-2,1],[6077.92,9E+09,9E+09,9E+09,9E+09,9E+09]],
                                        [[-17.6799,527.115,102.326],[0.938981,0.305706,0.151018,0.0453067],[-1,2,-2,1],[6076.76,9E+09,9E+09,9E+09,9E+09,9E+09]],
                                        [[-17.6731,527.982,102.957],[0.938608,0.306889,0.150913,0.0453823],[-1,2,-2,1],[6075.67,9E+09,9E+09,9E+09,9E+09,9E+09]],
                                        [[-17.6608,528.842,103.602],[0.938234,0.308074,0.150806,0.0454517],[-1,2,-2,1],[6074.65,9E+09,9E+09,9E+09,9E+09,9E+09]],
                                        [[-17.6528,529.703,104.249],[0.937852,0.309278,0.150694,0.0455123],[-1,2,-2,1],[6073.7,9E+09,9E+09,9E+09,9E+09,9E+09]],
                                        [[-17.6441,530.557,104.896],[0.937452,0.310536,0.150578,0.045584],[-1,2,-2,1],[6072.82,9E+09,9E+09,9E+09,9E+09,9E+09]],
                                        [[-17.6345,531.412,105.54],[0.937072,0.311732,0.150459,0.0456242],[-1,2,-2,1],[6072.01,9E+09,9E+09,9E+09,9E+09,9E+09]],
                                        [[-17.6243,532.263,106.189],[0.936701,0.312899,0.150339,0.0456555],[-1,2,-2,1],[6071.25,9E+09,9E+09,9E+09,9E+09,9E+09]],
                                        [[-17.6206,533.11,106.833],[0.936345,0.31402,0.150217,0.0456658],[-1,2,-2,1],[6070.55,9E+09,9E+09,9E+09,9E+09,9E+09]],
                                        [[-17.6145,533.947,107.488],[0.935988,0.31514,0.150092,0.045669],[-1,2,-2,1],[6069.9,9E+09,9E+09,9E+09,9E+09,9E+09]],
                                        [[-17.6089,534.792,108.116],[0.935646,0.316215,0.149966,0.0456526],[-1,2,-2,1],[6069.32,9E+09,9E+09,9E+09,9E+09,9E+09]],
                                        [[-17.6034,535.633,108.749],[0.935121,0.317188,0.151065,0.046044],[-1,2,-2,1],[6068.69,9E+09,9E+09,9E+09,9E+09,9E+09]],
                                        [[-17.594,536.482,109.383],[0.934605,0.31813,0.152159,0.0464155],[-1,2,-2,1],[6068.04,9E+09,9E+09,9E+09,9E+09,9E+09]],
                                        [[-17.583,537.332,110.035],[0.934107,0.319012,0.153255,0.0467815],[-1,2,-2,1],[6067.35,9E+09,9E+09,9E+09,9E+09,9E+09]],
                                        [[-17.5691,538.191,110.685],[0.933609,0.319885,0.154353,0.0471571],[-1,2,-2,1],[6066.63,9E+09,9E+09,9E+09,9E+09,9E+09]],
                                        [[-17.5532,539.041,111.347],[0.933119,0.320724,0.155452,0.0475303],[-1,2,-2,1],[6065.87,9E+09,9E+09,9E+09,9E+09,9E+09]],
                                        [[-17.5392,539.883,112.014],[0.932637,0.321529,0.156559,0.0479212],[-1,2,-2,1],[6065.1,9E+09,9E+09,9E+09,9E+09,9E+09]],
                                        [[-17.5267,540.735,112.676],[0.932161,0.322306,0.157671,0.0483258],[-1,2,-2,1],[6064.29,9E+09,9E+09,9E+09,9E+09,9E+09]],
                                        [[-17.5104,541.586,113.349],[0.931679,0.32308,0.158792,0.0487638],[-1,2,-2,1],[6063.44,9E+09,9E+09,9E+09,9E+09,9E+09]],
                                        [[-17.4956,542.427,114.025],[0.93121,0.323809,0.159921,0.0492138],[-1,2,-2,1],[6062.54,9E+09,9E+09,9E+09,9E+09,9E+09]],
                                        [[-17.4798,543.266,114.684],[0.930747,0.324504,0.161056,0.0496769],[-1,2,-2,1],[6061.62,9E+09,9E+09,9E+09,9E+09,9E+09]],
                                        [[-17.4642,544.094,115.363],[0.930275,0.325223,0.162187,0.050141],[-1,2,-2,1],[6060.65,9E+09,9E+09,9E+09,9E+09,9E+09]],
                                        [[-17.4548,544.916,116.055],[0.929797,0.325944,0.163324,0.0506324],[-1,2,-2,1],[6059.67,9E+09,9E+09,9E+09,9E+09,9E+09]],
                                        [[-17.4366,545.745,116.711],[0.929315,0.326668,0.164461,0.0511314],[-1,2,-2,1],[6058.64,9E+09,9E+09,9E+09,9E+09,9E+09]],
                                        [[-17.4275,546.583,117.363],[0.928818,0.327426,0.165596,0.051642],[-1,2,-2,1],[6057.57,9E+09,9E+09,9E+09,9E+09,9E+09]],
                                        [[-17.4142,547.414,118.016],[0.928323,0.328171,0.166732,0.0521603],[-1,2,-2,1],[6056.45,9E+09,9E+09,9E+09,9E+09,9E+09]],
                                        [[-17.3987,548.247,118.675],[0.927831,0.328891,0.167878,0.0527008],[-1,2,-2,1],[6055.29,9E+09,9E+09,9E+09,9E+09,9E+09]],
                                        [[-17.3829,549.073,119.331],[0.927314,0.329664,0.16903,0.0532886],[-1,2,-2,1],[6054.1,9E+09,9E+09,9E+09,9E+09,9E+09]],
                                        [[-17.3691,549.899,119.989],[0.926793,0.330433,0.170187,0.0538971],[-1,2,-2,1],[6052.88,9E+09,9E+09,9E+09,9E+09,9E+09]],
                                        [[-17.348,550.724,120.653],[0.926271,0.331189,0.171354,0.0545345],[-1,2,-2,1],[6051.61,9E+09,9E+09,9E+09,9E+09,9E+09]],
                                        [[-17.3326,551.544,121.318],[0.925746,0.331938,0.172527,0.0551949],[-1,2,-2,1],[6050.3,9E+09,9E+09,9E+09,9E+09,9E+09]],
                                        [[-17.317,552.356,121.993],[0.925211,0.3327,0.173705,0.0558807],[-1,2,-2,1],[6048.96,9E+09,9E+09,9E+09,9E+09,9E+09]],
                                        [[-17.3042,553.172,122.671],[0.924677,0.333445,0.174887,0.0565785],[-1,2,-2,1],[6047.58,9E+09,9E+09,9E+09,9E+09,9E+09]],
                                        [[-17.2941,553.987,123.348],[0.924135,0.334201,0.176072,0.0572948],[-1,2,-2,1],[6046.16,9E+09,9E+09,9E+09,9E+09,9E+09]],
                                        [[-17.2805,554.799,124.017],[0.92358,0.334984,0.177255,0.0580201],[-1,2,-2,1],[6044.7,9E+09,9E+09,9E+09,9E+09,9E+09]],
                                        [[-17.2733,555.601,124.697],[0.923025,0.335756,0.17844,0.0587561],[-1,2,-2,1],[6043.2,9E+09,9E+09,9E+09,9E+09,9E+09]],
                                        [[-17.2647,556.406,125.369],[0.922469,0.336526,0.17962,0.0594803],[-1,2,-2,1],[6041.67,9E+09,9E+09,9E+09,9E+09,9E+09]],
                                        [[-17.254,557.216,126.037],[0.921883,0.337375,0.180787,0.0602094],[-1,2,-2,1],[6040.1,9E+09,9E+09,9E+09,9E+09,9E+09]],
                                        [[-17.2408,558.009,126.717],[0.921288,0.338244,0.181949,0.0609354],[-1,2,-2,1],[6038.51,9E+09,9E+09,9E+09,9E+09,9E+09]],
                                        [[-17.2339,558.804,127.382],[0.920671,0.339174,0.183098,0.0616583],[-1,2,-2,1],[6036.91,9E+09,9E+09,9E+09,9E+09,9E+09]],
                                        [[-17.2205,559.596,128.054],[0.92001,0.340207,0.18424,0.0624151],[-1,2,-2,1],[6035.28,9E+09,9E+09,9E+09,9E+09,9E+09]],
                                        [[-17.2075,560.378,128.736],[0.919333,0.341281,0.185373,0.0631688],[-1,2,-2,1],[6033.64,9E+09,9E+09,9E+09,9E+09,9E+09]],
                                        [[-17.196,561.181,129.406],[0.918653,0.342348,0.186508,0.0639368],[-1,2,-2,1],[6032,9E+09,9E+09,9E+09,9E+09,9E+09]],
                                        [[-17.184,561.978,130.071],[0.917967,0.343425,0.18764,0.0647051],[-1,2,-2,1],[6030.32,9E+09,9E+09,9E+09,9E+09,9E+09]],
                                        [[-17.1775,562.764,130.761],[0.91728,0.344497,0.188767,0.0654685],[-1,2,-2,1],[6028.63,9E+09,9E+09,9E+09,9E+09,9E+09]],
                                        [[-17.1652,563.545,131.445],[0.916597,0.345553,0.189891,0.0662198],[-1,2,-2,1],[6026.94,9E+09,9E+09,9E+09,9E+09,9E+09]],
                                        [[-17.1556,564.325,132.132],[0.91591,0.346613,0.191008,0.0669644],[-1,2,-2,1],[6025.24,9E+09,9E+09,9E+09,9E+09,9E+09]],
                                        [[-17.1472,565.105,132.821],[0.915229,0.347662,0.192112,0.067675],[-1,2,-2,1],[6023.54,9E+09,9E+09,9E+09,9E+09,9E+09]],
                                        [[-17.14,565.882,133.514],[0.914546,0.348715,0.193206,0.0683669],[-1,2,-2,1],[6021.83,9E+09,9E+09,9E+09,9E+09,9E+09]],
                                        [[-17.1329,566.663,134.208],[0.913849,0.349802,0.194293,0.069062],[-1,2,-2,1],[6020.12,9E+09,9E+09,9E+09,9E+09,9E+09]],
                                        [[-17.1288,567.444,134.904],[0.91313,0.350942,0.195367,0.0697547],[-1,2,-2,1],[6018.4,9E+09,9E+09,9E+09,9E+09,9E+09]],
                                        [[-17.1189,568.226,135.6],[0.912407,0.35208,0.19644,0.0704533],[-1,2,-2,1],[6016.68,9E+09,9E+09,9E+09,9E+09,9E+09]],
                                        [[-17.1108,569.01,136.296],[0.911695,0.353187,0.197509,0.0711369],[-1,2,-2,1],[6014.96,9E+09,9E+09,9E+09,9E+09,9E+09]],
                                        [[-17.0979,569.793,136.993],[0.910981,0.35429,0.198578,0.0718257],[-1,2,-2,1],[6013.23,9E+09,9E+09,9E+09,9E+09,9E+09]],
                                        [[-17.0845,570.563,137.715],[0.910275,0.355362,0.199648,0.0725106],[-1,2,-2,1],[6011.5,9E+09,9E+09,9E+09,9E+09,9E+09]],
                                        [[-17.0735,571.34,138.427],[0.909574,0.356415,0.200714,0.0731881],[-1,2,-2,1],[6009.78,9E+09,9E+09,9E+09,9E+09,9E+09]],
                                        [[-17.0594,572.108,139.147],[0.90887,0.357477,0.201772,0.0738515],[-1,2,-2,1],[6008.05,9E+09,9E+09,9E+09,9E+09,9E+09]],
                                        [[-17.0492,572.877,139.863],[0.908169,0.358518,0.202831,0.0745213],[-1,2,-2,1],[6006.32,9E+09,9E+09,9E+09,9E+09,9E+09]],
                                        [[-17.0394,573.644,140.593],[0.907486,0.359508,0.203891,0.0751743],[-1,2,-2,1],[6004.59,9E+09,9E+09,9E+09,9E+09,9E+09]],
                                        [[-17.0297,574.412,141.321],[0.906798,0.360506,0.204945,0.0758252],[-1,2,-2,1],[6002.86,9E+09,9E+09,9E+09,9E+09,9E+09]],
                                        [[-17.0186,575.176,142.052],[0.90614,0.361425,0.206003,0.0764531],[-1,2,-2,1],[6001.11,9E+09,9E+09,9E+09,9E+09,9E+09]],
                                        [[-17.0088,575.944,142.776],[0.905504,0.362286,0.207061,0.0770613],[-1,2,-2,1],[5999.36,9E+09,9E+09,9E+09,9E+09,9E+09]],
                                        [[-16.9983,576.717,143.508],[0.904872,0.363124,0.208121,0.0776731],[-1,2,-2,1],[5997.59,9E+09,9E+09,9E+09,9E+09,9E+09]],
                                        [[-16.9863,577.477,144.239],[0.904258,0.363922,0.209176,0.0782555],[-1,2,-2,1],[5995.81,9E+09,9E+09,9E+09,9E+09,9E+09]],
                                        [[-16.9737,578.242,144.972],[0.903642,0.364726,0.210222,0.0788226],[-1,2,-2,1],[5994.04,9E+09,9E+09,9E+09,9E+09,9E+09]],
                                        [[-16.9602,579.003,145.71],[0.903032,0.365512,0.211264,0.079379],[-1,2,-2,1],[5992.25,9E+09,9E+09,9E+09,9E+09,9E+09]],
                                        [[-16.9522,579.762,146.453],[0.90243,0.366272,0.212309,0.0799348],[-1,2,-2,1],[5990.46,9E+09,9E+09,9E+09,9E+09,9E+09]],
                                        [[-16.9384,580.517,147.209],[0.901832,0.367015,0.213355,0.0804935],[-1,2,-2,1],[5988.66,9E+09,9E+09,9E+09,9E+09,9E+09]],
                                        [[-16.9285,581.274,147.953],[0.901241,0.367728,0.214407,0.0810602],[-1,2,-2,1],[5986.86,9E+09,9E+09,9E+09,9E+09,9E+09]],
                                        [[-16.9173,582.041,148.689],[0.900662,0.368401,0.215465,0.0816282],[-1,2,-2,1],[5985.03,9E+09,9E+09,9E+09,9E+09,9E+09]],
                                        [[-16.9042,582.801,149.429],[0.900102,0.369022,0.216528,0.0821877],[-1,2,-2,1],[5983.18,9E+09,9E+09,9E+09,9E+09,9E+09]],
                                        [[-16.8914,583.563,150.169],[0.899573,0.369565,0.217595,0.0827223],[-1,2,-2,1],[5981.32,9E+09,9E+09,9E+09,9E+09,9E+09]],
                                        [[-16.8783,584.325,150.925],[0.899036,0.370125,0.218657,0.0832571],[-1,2,-2,1],[5979.43,9E+09,9E+09,9E+09,9E+09,9E+09]],
                                        [[-16.8636,585.083,151.681],[0.898499,0.370681,0.219716,0.0837891],[-1,2,-2,1],[5977.54,9E+09,9E+09,9E+09,9E+09,9E+09]],
                                        [[-16.8514,585.836,152.437],[0.897951,0.371259,0.220771,0.0843248],[-1,2,-2,1],[5975.64,9E+09,9E+09,9E+09,9E+09,9E+09]],
                                        [[-16.8405,586.601,153.176],[0.897402,0.371837,0.221824,0.0848631],[-1,2,-2,1],[5973.73,9E+09,9E+09,9E+09,9E+09,9E+09]],
                                        [[-16.8295,587.356,153.931],[0.896843,0.372432,0.222874,0.0854085],[-1,2,-2,1],[5971.79,9E+09,9E+09,9E+09,9E+09,9E+09]],
                                        [[-16.8167,588.115,154.681],[0.896279,0.373032,0.223923,0.0859605],[-1,2,-2,1],[5969.85,9E+09,9E+09,9E+09,9E+09,9E+09]],
                                        [[-16.8037,588.871,155.438],[0.895704,0.373653,0.22497,0.0865257],[-1,2,-2,1],[5967.89,9E+09,9E+09,9E+09,9E+09,9E+09]],
                                        [[-16.7905,589.632,156.19],[0.895131,0.374261,0.226018,0.0870912],[-1,2,-2,1],[5965.92,9E+09,9E+09,9E+09,9E+09,9E+09]],
                                        [[-16.7731,590.388,156.946],[0.894558,0.374865,0.227064,0.0876579],[-1,2,-2,1],[5963.94,9E+09,9E+09,9E+09,9E+09,9E+09]],
                                        [[-16.7538,591.136,157.709],[0.893985,0.375459,0.228114,0.0882334],[-1,2,-2,1],[5961.94,9E+09,9E+09,9E+09,9E+09,9E+09]],
                                        [[-16.7362,591.886,158.469],[0.893402,0.376062,0.229169,0.0888335],[-1,2,-2,1],[5959.94,9E+09,9E+09,9E+09,9E+09,9E+09]],
                                        [[-16.7208,592.629,159.228],[0.892808,0.376682,0.230223,0.0894495],[-1,2,-2,1],[5957.94,9E+09,9E+09,9E+09,9E+09,9E+09]],
                                        [[-16.7054,593.379,159.993],[0.892206,0.377296,0.231294,0.0901117],[-1,2,-2,1],[5955.94,9E+09,9E+09,9E+09,9E+09,9E+09]],
                                        [[-16.6891,594.121,160.759],[0.891586,0.377928,0.232373,0.0908148],[-1,2,-2,1],[5953.94,9E+09,9E+09,9E+09,9E+09,9E+09]],
                                        [[-16.6767,594.866,161.521],[0.890947,0.378578,0.233467,0.0915759],[-1,2,-2,1],[5951.94,9E+09,9E+09,9E+09,9E+09,9E+09]],
                                        [[-16.6599,595.61,162.28],[0.89031,0.379197,0.234577,0.0923686],[-1,2,-2,1],[5949.94,9E+09,9E+09,9E+09,9E+09,9E+09]],
                                        [[-16.6445,596.358,163.028],[0.889663,0.379817,0.235697,0.0931954],[-1,2,-2,1],[5947.94,9E+09,9E+09,9E+09,9E+09,9E+09]],
                                        [[-16.6301,597.099,163.794],[0.889016,0.380423,0.236825,0.0940401],[-1,2,-2,1],[5945.94,9E+09,9E+09,9E+09,9E+09,9E+09]],
                                        [[-16.6141,597.828,164.572],[0.888358,0.381037,0.237956,0.0949066],[-1,2,-2,1],[5943.94,9E+09,9E+09,9E+09,9E+09,9E+09]],
                                        [[-16.6011,598.559,165.344],[0.887682,0.381676,0.239092,0.0958056],[-1,2,-2,1],[5941.94,9E+09,9E+09,9E+09,9E+09,9E+09]],
                                        [[-16.5855,599.286,166.119],[0.886988,0.382334,0.240236,0.0967462],[-1,2,-2,1],[5939.94,9E+09,9E+09,9E+09,9E+09,9E+09]],
                                        [[-16.5693,600.014,166.886],[0.886286,0.382987,0.241391,0.0977185],[-1,2,-2,1],[5937.94,9E+09,9E+09,9E+09,9E+09,9E+09]],
                                        [[-16.5532,600.739,167.655],[0.885573,0.383639,0.242558,0.098729],[-1,2,-2,1],[5935.94,9E+09,9E+09,9E+09,9E+09,9E+09]],
                                        [[-16.5396,601.461,168.425],[0.884851,0.384296,0.243728,0.0997577],[-1,2,-2,1],[5933.94,9E+09,9E+09,9E+09,9E+09,9E+09]],
                                        [[-16.5225,602.177,169.19],[0.884119,0.384961,0.244901,0.100806],[-1,2,-2,1],[5931.94,9E+09,9E+09,9E+09,9E+09,9E+09]],
                                        [[-16.5056,602.891,169.951],[0.883375,0.385634,0.24608,0.10188],[-1,2,-2,1],[5929.94,9E+09,9E+09,9E+09,9E+09,9E+09]],
                                        [[-16.4928,603.604,170.711],[0.882627,0.386304,0.24726,0.102963],[-1,2,-2,1],[5927.94,9E+09,9E+09,9E+09,9E+09,9E+09]],
                                        [[-16.4845,604.311,171.477],[0.881863,0.387006,0.248432,0.10405],[-1,2,-2,1],[5925.94,9E+09,9E+09,9E+09,9E+09,9E+09]],
                                        [[-16.4734,605.012,172.239],[0.881096,0.387702,0.249604,0.10514],[-1,2,-2,1],[5923.94,9E+09,9E+09,9E+09,9E+09,9E+09]],
